LIN {X -45.187,Y 28.575,Z -129.329,A 90.000,B 90.000,C 0.000} C_DIS
LIN {X -45.416,Y 28.575,Z -128.828,A 90.000,B 90.000,C 0.000} C_DIS
LIN {X -45.639,Y 28.575,Z -128.325,A 90.000,B 90.000,C 0.000} C_DIS
LIN {X -46.722,Y 28.575,Z -126.161,A 90.000,B 90.000,C 0.000} C_DIS
LIN {X -47.769,Y 28.575,Z -123.979,A 90.000,B 90.000,C 0.000} C_DIS
LIN {X -48.781,Y 28.575,Z -121.781,A 90.000,B 90.000,C 0.000} C_DIS
LIN {X -144.015,Y 28.575,Z -121.781,A 90.000,B 90.000,C 0.000} C_DIS
LIN {X -144.015,Y 28.575,Z -114.232,A 90.000,B 90.000,C 0.000} C_DIS
LIN {X -53.262,Y 28.575,Z -114.232,A 90.000,B 90.000,C 0.000} C_DIS
LIN {X -53.882,Y 28.575,Z -113.422,A 90.000,B 90.000,C 0.000} C_DIS
LIN {X -54.518,Y 28.575,Z -112.624,A 90.000,B 90.000,C 0.000} C_DIS
LIN {X -56.238,Y 28.575,Z -110.408,A 90.000,B 90.000,C 0.000} C_DIS
LIN {X -57.937,Y 28.575,Z -108.176,A 90.000,B 90.000,C 0.000} C_DIS
LIN {X -59.127,Y 28.575,Z -106.683,A 90.000,B 90.000,C 0.000} C_DIS
LIN {X -144.015,Y 28.575,Z -106.683,A 90.000,B 90.000,C 0.000} C_DIS
LIN {X -144.015,Y 28.575,Z -99.134,A 90.000,B 90.000,C 0.000} C_DIS
LIN {X -64.843,Y 28.575,Z -99.134,A 90.000,B 90.000,C 0.000} C_DIS
LIN {X -65.709,Y 28.575,Z -97.932,A 90.000,B 90.000,C 0.000} C_DIS
LIN {X -66.964,Y 28.575,Z -96.315,A 90.000,B 90.000,C 0.000} C_DIS
LIN {X -68.244,Y 28.575,Z -94.718,A 90.000,B 90.000,C 0.000} C_DIS
LIN {X -69.549,Y 28.575,Z -93.142,A 90.000,B 90.000,C 0.000} C_DIS
LIN {X -70.879,Y 28.575,Z -91.586,A 90.000,B 90.000,C 0.000} C_DIS
LIN {X -144.015,Y 28.575,Z -91.586,A 90.000,B 90.000,C 0.000} C_DIS
LIN {X -144.015,Y 28.575,Z -84.037,A 90.000,B 90.000,C 0.000} C_DIS
LIN {X -77.937,Y 28.575,Z -84.037,A 90.000,B 90.000,C 0.000} C_DIS
LIN {X -78.622,Y 28.575,Z -83.298,A 90.000,B 90.000,C 0.000} C_DIS
LIN {X -79.761,Y 28.575,Z -83.093,A 90.000,B 90.000,C 0.000} C_DIS
LIN {X -80.886,Y 28.575,Z -82.817,A 90.000,B 90.000,C 0.000} C_DIS
LIN {X -81.990,Y 28.575,Z -82.470,A 90.000,B 90.000,C 0.000} C_DIS
LIN {X -83.070,Y 28.575,Z -82.054,A 90.000,B 90.000,C 0.000} C_DIS
LIN {X -84.122,Y 28.575,Z -81.570,A 90.000,B 90.000,C 0.000} C_DIS
LIN {X -85.141,Y 28.575,Z -81.021,A 90.000,B 90.000,C 0.000} C_DIS
LIN {X -86.123,Y 28.575,Z -80.408,A 90.000,B 90.000,C 0.000} C_DIS
LIN {X -87.065,Y 28.575,Z -79.735,A 90.000,B 90.000,C 0.000} C_DIS
LIN {X -87.961,Y 28.575,Z -79.003,A 90.000,B 90.000,C 0.000} C_DIS
LIN {X -88.810,Y 28.575,Z -78.215,A 90.000,B 90.000,C 0.000} C_DIS
LIN {X -89.608,Y 28.575,Z -77.376,A 90.000,B 90.000,C 0.000} C_DIS
LIN {X -90.350,Y 28.575,Z -76.488,A 90.000,B 90.000,C 0.000} C_DIS
LIN {X -144.015,Y 28.575,Z -76.488,A 90.000,B 90.000,C 0.000} C_DIS
LIN {X -144.015,Y 28.575,Z -68.939,A 90.000,B 90.000,C 0.000} C_DIS
LIN {X -94.422,Y 28.575,Z -68.939,A 90.000,B 90.000,C 0.000} C_DIS
LIN {X -95.090,Y 28.575,Z -68.358,A 90.000,B 90.000,C 0.000} C_DIS
LIN {X -95.244,Y 28.575,Z -68.214,A 90.000,B 90.000,C 0.000} C_DIS
LIN {X -95.839,Y 28.575,Z -67.609,A 90.000,B 90.000,C 0.000} C_DIS
LIN {X -96.393,Y 28.575,Z -66.968,A 90.000,B 90.000,C 0.000} C_DIS
LIN {X -96.906,Y 28.575,Z -66.291,A 90.000,B 90.000,C 0.000} C_DIS
LIN {X -97.373,Y 28.575,Z -65.584,A 90.000,B 90.000,C 0.000} C_DIS
LIN {X -97.795,Y 28.575,Z -64.848,A 90.000,B 90.000,C 0.000} C_DIS
LIN {X -98.168,Y 28.575,Z -64.086,A 90.000,B 90.000,C 0.000} C_DIS
LIN {X -99.173,Y 28.575,Z -63.219,A 90.000,B 90.000,C 0.000} C_DIS
LIN {X -100.151,Y 28.575,Z -62.320,A 90.000,B 90.000,C 0.000} C_DIS
LIN {X -101.099,Y 28.575,Z -61.390,A 90.000,B 90.000,C 0.000} C_DIS
LIN {X -144.015,Y 28.575,Z -61.390,A 90.000,B 90.000,C 0.000} C_DIS
LIN {X -144.015,Y 28.575,Z -53.842,A 90.000,B 90.000,C 0.000} C_DIS
LIN {X -106.042,Y 28.575,Z -53.842,A 90.000,B 90.000,C 0.000} C_DIS
LIN {X -106.315,Y 28.575,Z -52.946,A 90.000,B 90.000,C 0.000} C_DIS
LIN {X -106.538,Y 28.575,Z -52.036,A 90.000,B 90.000,C 0.000} C_DIS
LIN {X -106.713,Y 28.575,Z -51.115,A 90.000,B 90.000,C 0.000} C_DIS
LIN {X -106.837,Y 28.575,Z -50.186,A 90.000,B 90.000,C 0.000} C_DIS
LIN {X -106.910,Y 28.575,Z -49.252,A 90.000,B 90.000,C 0.000} C_DIS
LIN {X -106.883,Y 28.575,Z -48.505,A 90.000,B 90.000,C 0.000} C_DIS
LIN {X -106.812,Y 28.575,Z -47.761,A 90.000,B 90.000,C 0.000} C_DIS
LIN {X -106.696,Y 28.575,Z -47.023,A 90.000,B 90.000,C 0.000} C_DIS
LIN {X -106.537,Y 28.575,Z -46.293,A 90.000,B 90.000,C 0.000} C_DIS
LIN {X -144.015,Y 28.575,Z -46.293,A 90.000,B 90.000,C 0.000} C_DIS
LIN {X -144.015,Y 28.575,Z -38.744,A 90.000,B 90.000,C 0.000} C_DIS
LIN {X -101.192,Y 28.575,Z -38.744,A 90.000,B 90.000,C 0.000} C_DIS
LIN {X -144.015,Y 28.575,Z -31.195,A 90.000,B 90.000,C 0.000} C_DIS
LIN {X 98.089,Y 28.575,Z -31.195,A 90.000,B 90.000,C 0.000} C_DIS
LIN {X 99.517,Y 28.575,Z -30.557,A 90.000,B 90.000,C 0.000} C_DIS
LIN {X 100.960,Y 28.575,Z -29.954,A 90.000,B 90.000,C 0.000} C_DIS
LIN {X 102.417,Y 28.575,Z -29.386,A 90.000,B 90.000,C 0.000} C_DIS
LIN {X 103.674,Y 28.575,Z -28.880,A 90.000,B 90.000,C 0.000} C_DIS
LIN {X 104.953,Y 28.575,Z -28.431,A 90.000,B 90.000,C 0.000} C_DIS
LIN {X 106.251,Y 28.575,Z -28.040,A 90.000,B 90.000,C 0.000} C_DIS
LIN {X 107.565,Y 28.575,Z -27.708,A 90.000,B 90.000,C 0.000} C_DIS
LIN {X 108.892,Y 28.575,Z -27.435,A 90.000,B 90.000,C 0.000} C_DIS
LIN {X 109.865,Y 28.575,Z -27.357,A 90.000,B 90.000,C 0.000} C_DIS
LIN {X 110.841,Y 28.575,Z -27.343,A 90.000,B 90.000,C 0.000} C_DIS
LIN {X 111.816,Y 28.575,Z -27.395,A 90.000,B 90.000,C 0.000} C_DIS
LIN {X 112.785,Y 28.575,Z -27.512,A 90.000,B 90.000,C 0.000} C_DIS
LIN {X 113.744,Y 28.575,Z -27.693,A 90.000,B 90.000,C 0.000} C_DIS
LIN {X 114.689,Y 28.575,Z -27.938,A 90.000,B 90.000,C 0.000} C_DIS
LIN {X 114.871,Y 28.575,Z -27.996,A 90.000,B 90.000,C 0.000} C_DIS
LIN {X 115.775,Y 28.575,Z -28.294,A 90.000,B 90.000,C 0.000} C_DIS
LIN {X 116.659,Y 28.575,Z -28.648,A 90.000,B 90.000,C 0.000} C_DIS
LIN {X 117.519,Y 28.575,Z -29.056,A 90.000,B 90.000,C 0.000} C_DIS
LIN {X 118.352,Y 28.575,Z -29.518,A 90.000,B 90.000,C 0.000} C_DIS
LIN {X 118.488,Y 28.575,Z -29.602,A 90.000,B 90.000,C 0.000} C_DIS
LIN {X 119.234,Y 28.575,Z -30.088,A 90.000,B 90.000,C 0.000} C_DIS
LIN {X 119.949,Y 28.575,Z -30.620,A 90.000,B 90.000,C 0.000} C_DIS
LIN {X 120.629,Y 28.575,Z -31.195,A 90.000,B 90.000,C 0.000} C_DIS
LIN {X 144.015,Y 28.575,Z -31.195,A 90.000,B 90.000,C 0.000} C_DIS
LIN {X 144.015,Y 28.575,Z -38.744,A 90.000,B 90.000,C 0.000} C_DIS
LIN {X 125.030,Y 28.575,Z -38.744,A 90.000,B 90.000,C 0.000} C_DIS
LIN {X 125.175,Y 28.575,Z -39.493,A 90.000,B 90.000,C 0.000} C_DIS
LIN {X 125.280,Y 28.575,Z -40.248,A 90.000,B 90.000,C 0.000} C_DIS
LIN {X 125.344,Y 28.575,Z -41.008,A 90.000,B 90.000,C 0.000} C_DIS
LIN {X 125.413,Y 28.575,Z -42.067,A 90.000,B 90.000,C 0.000} C_DIS
LIN {X 125.426,Y 28.575,Z -43.127,A 90.000,B 90.000,C 0.000} C_DIS
LIN {X 125.383,Y 28.575,Z -44.187,A 90.000,B 90.000,C 0.000} C_DIS
LIN {X 125.285,Y 28.575,Z -45.243,A 90.000,B 90.000,C 0.000} C_DIS
LIN {X 125.131,Y 28.575,Z -46.293,A 90.000,B 90.000,C 0.000} C_DIS
LIN {X 144.015,Y 28.575,Z -46.293,A 90.000,B 90.000,C 0.000} C_DIS
LIN {X 144.015,Y 28.575,Z -53.842,A 90.000,B 90.000,C 0.000} C_DIS
LIN {X 122.274,Y 28.575,Z -53.842,A 90.000,B 90.000,C 0.000} C_DIS
LIN {X 121.422,Y 28.575,Z -55.612,A 90.000,B 90.000,C 0.000} C_DIS
LIN {X 120.619,Y 28.575,Z -57.405,A 90.000,B 90.000,C 0.000} C_DIS
LIN {X 119.868,Y 28.575,Z -59.220,A 90.000,B 90.000,C 0.000} C_DIS
LIN {X 119.167,Y 28.575,Z -61.055,A 90.000,B 90.000,C 0.000} C_DIS
LIN {X 119.069,Y 28.575,Z -61.390,A 90.000,B 90.000,C 0.000} C_DIS
LIN {X 144.015,Y 28.575,Z -61.390,A 90.000,B 90.000,C 0.000} C_DIS
LIN {X 144.015,Y 28.575,Z -68.939,A 90.000,B 90.000,C 0.000} C_DIS
LIN {X 116.890,Y 28.575,Z -68.939,A 90.000,B 90.000,C 0.000} C_DIS
LIN {X 116.236,Y 28.575,Z -70.854,A 90.000,B 90.000,C 0.000} C_DIS
LIN {X 115.531,Y 28.575,Z -72.752,A 90.000,B 90.000,C 0.000} C_DIS
LIN {X 114.777,Y 28.575,Z -74.630,A 90.000,B 90.000,C 0.000} C_DIS
LIN {X 113.973,Y 28.575,Z -76.488,A 90.000,B 90.000,C 0.000} C_DIS
LIN {X 144.015,Y 28.575,Z -76.488,A 90.000,B 90.000,C 0.000} C_DIS
LIN {X 144.015,Y 28.575,Z -84.037,A 90.000,B 90.000,C 0.000} C_DIS
LIN {X 110.073,Y 28.575,Z -84.037,A 90.000,B 90.000,C 0.000} C_DIS
LIN {X 109.299,Y 28.575,Z -85.323,A 90.000,B 90.000,C 0.000} C_DIS
LIN {X 108.499,Y 28.575,Z -86.594,A 90.000,B 90.000,C 0.000} C_DIS
LIN {X 107.675,Y 28.575,Z -87.849,A 90.000,B 90.000,C 0.000} C_DIS
LIN {X 107.763,Y 28.575,Z -89.093,A 90.000,B 90.000,C 0.000} C_DIS
LIN {X 107.830,Y 28.575,Z -90.339,A 90.000,B 90.000,C 0.000} C_DIS
LIN {X 107.876,Y 28.575,Z -91.586,A 90.000,B 90.000,C 0.000} C_DIS
LIN {X 144.015,Y 28.575,Z -91.586,A 90.000,B 90.000,C 0.000} C_DIS
LIN {X 144.015,Y 28.575,Z -99.134,A 90.000,B 90.000,C 0.000} C_DIS
LIN {X 107.706,Y 28.575,Z -99.134,A 90.000,B 90.000,C 0.000} C_DIS
LIN {X 107.629,Y 28.575,Z -100.093,A 90.000,B 90.000,C 0.000} C_DIS
LIN {X 107.540,Y 28.575,Z -101.051,A 90.000,B 90.000,C 0.000} C_DIS
LIN {X 107.480,Y 28.575,Z -102.572,A 90.000,B 90.000,C 0.000} C_DIS
LIN {X 107.467,Y 28.575,Z -102.703,A 90.000,B 90.000,C 0.000} C_DIS
LIN {X 107.463,Y 28.575,Z -103.506,A 90.000,B 90.000,C 0.000} C_DIS
LIN {X 107.504,Y 28.575,Z -104.308,A 90.000,B 90.000,C 0.000} C_DIS
LIN {X 107.589,Y 28.575,Z -105.106,A 90.000,B 90.000,C 0.000} C_DIS
LIN {X 107.718,Y 28.575,Z -105.899,A 90.000,B 90.000,C 0.000} C_DIS
LIN {X 107.891,Y 28.575,Z -106.683,A 90.000,B 90.000,C 0.000} C_DIS
LIN {X 144.015,Y 28.575,Z -106.683,A 90.000,B 90.000,C 0.000} C_DIS
LIN {X 144.015,Y 28.575,Z -114.232,A 90.000,B 90.000,C 0.000} C_DIS
LIN {X 108.666,Y 28.575,Z -114.232,A 90.000,B 90.000,C 0.000} C_DIS
LIN {X 108.827,Y 28.575,Z -116.746,A 90.000,B 90.000,C 0.000} C_DIS
LIN {X 108.950,Y 28.575,Z -119.263,A 90.000,B 90.000,C 0.000} C_DIS
LIN {X 109.037,Y 28.575,Z -121.781,A 90.000,B 90.000,C 0.000} C_DIS
LIN {X 144.015,Y 28.575,Z -121.781,A 90.000,B 90.000,C 0.000} C_DIS
LIN {X 144.015,Y 28.575,Z -129.329,A 90.000,B 90.000,C 0.000} C_DIS
LIN {X 109.075,Y 28.575,Z -129.329,A 90.000,B 90.000,C 0.000} C_DIS
LIN {X 109.014,Y 28.575,Z -131.847,A 90.000,B 90.000,C 0.000} C_DIS
LIN {X 108.916,Y 28.575,Z -134.363,A 90.000,B 90.000,C 0.000} C_DIS
LIN {X 108.782,Y 28.575,Z -136.878,A 90.000,B 90.000,C 0.000} C_DIS
LIN {X 144.015,Y 28.575,Z -136.878,A 90.000,B 90.000,C 0.000} C_DIS
LIN {X 144.015,Y 28.575,Z -144.427,A 90.000,B 90.000,C 0.000} C_DIS
LIN {X 108.182,Y 28.575,Z -144.427,A 90.000,B 90.000,C 0.000} C_DIS
LIN {X 107.856,Y 28.575,Z -148.203,A 90.000,B 90.000,C 0.000} C_DIS
LIN {X 107.490,Y 28.575,Z -151.976,A 90.000,B 90.000,C 0.000} C_DIS
LIN {X 144.015,Y 28.575,Z -151.976,A 90.000,B 90.000,C 0.000} C_DIS
LIN {X 144.015,Y 28.575,Z -159.525,A 90.000,B 90.000,C 0.000} C_DIS
LIN {X 106.632,Y 28.575,Z -159.525,A 90.000,B 90.000,C 0.000} C_DIS
LIN {X 106.141,Y 28.575,Z -163.302,A 90.000,B 90.000,C 0.000} C_DIS
LIN {X 105.608,Y 28.575,Z -167.073,A 90.000,B 90.000,C 0.000} C_DIS
LIN {X 144.015,Y 28.575,Z -167.073,A 90.000,B 90.000,C 0.000} C_DIS
LIN {X 144.015,Y 28.575,Z -174.622,A 90.000,B 90.000,C 0.000} C_DIS
LIN {X 104.436,Y 28.575,Z -174.622,A 90.000,B 90.000,C 0.000} C_DIS
LIN {X 104.078,Y 28.575,Z -177.133,A 90.000,B 90.000,C 0.000} C_DIS
LIN {X 103.757,Y 28.575,Z -179.650,A 90.000,B 90.000,C 0.000} C_DIS
LIN {X 103.474,Y 28.575,Z -182.171,A 90.000,B 90.000,C 0.000} C_DIS
LIN {X 144.015,Y 28.575,Z -182.171,A 90.000,B 90.000,C 0.000} C_DIS
LIN {X 144.015,Y 28.575,Z -189.720,A 90.000,B 90.000,C 0.000} C_DIS
LIN {X 102.854,Y 28.575,Z -189.720,A 90.000,B 90.000,C 0.000} C_DIS
LIN {X 102.786,Y 28.575,Z -190.930,A 90.000,B 90.000,C 0.000} C_DIS
LIN {X 102.727,Y 28.575,Z -192.140,A 90.000,B 90.000,C 0.000} C_DIS
LIN {X 102.588,Y 28.575,Z -193.853,A 90.000,B 90.000,C 0.000} C_DIS
LIN {X 102.412,Y 28.575,Z -195.563,A 90.000,B 90.000,C 0.000} C_DIS
LIN {X 102.197,Y 28.575,Z -197.269,A 90.000,B 90.000,C 0.000} C_DIS
LIN {X 144.015,Y 28.575,Z -197.269,A 90.000,B 90.000,C 0.000} C_DIS
LIN {X 144.015,Y 28.575,Z -204.817,A 90.000,B 90.000,C 0.000} C_DIS
LIN {X 100.774,Y 28.575,Z -204.817,A 90.000,B 90.000,C 0.000} C_DIS
LIN {X 100.506,Y 28.575,Z -205.895,A 90.000,B 90.000,C 0.000} C_DIS
LIN {X 100.223,Y 28.575,Z -206.969,A 90.000,B 90.000,C 0.000} C_DIS
LIN {X 99.604,Y 28.575,Z -209.358,A 90.000,B 90.000,C 0.000} C_DIS
LIN {X 99.003,Y 28.575,Z -211.751,A 90.000,B 90.000,C 0.000} C_DIS
LIN {X 98.837,Y 28.575,Z -212.366,A 90.000,B 90.000,C 0.000} C_DIS
LIN {X 144.015,Y 28.575,Z -212.366,A 90.000,B 90.000,C 0.000} C_DIS
LIN {X 144.015,Y 28.575,Z -219.915,A 90.000,B 90.000,C 0.000} C_DIS
LIN {X 96.861,Y 28.575,Z -219.915,A 90.000,B 90.000,C 0.000} C_DIS
LIN {X 95.882,Y 28.575,Z -223.687,A 90.000,B 90.000,C 0.000} C_DIS
LIN {X 94.920,Y 28.575,Z -227.464,A 90.000,B 90.000,C 0.000} C_DIS
LIN {X 144.015,Y 28.575,Z -227.464,A 90.000,B 90.000,C 0.000} C_DIS
LIN {X 144.015,Y 28.575,Z -235.012,A 90.000,B 90.000,C 0.000} C_DIS
LIN {X 92.952,Y 28.575,Z -235.012,A 90.000,B 90.000,C 0.000} C_DIS
LIN {X 92.216,Y 28.575,Z -237.541,A 90.000,B 90.000,C 0.000} C_DIS
LIN {X 91.439,Y 28.575,Z -240.057,A 90.000,B 90.000,C 0.000} C_DIS
LIN {X 90.622,Y 28.575,Z -242.561,A 90.000,B 90.000,C 0.000} C_DIS
LIN {X 144.015,Y 28.575,Z -242.561,A 90.000,B 90.000,C 0.000} C_DIS
LIN {X 144.015,Y 28.575,Z -23.646,A 90.000,B 90.000,C 0.000} C_DIS
LIN {X -144.015,Y 28.575,Z -23.646,A 90.000,B 90.000,C 0.000} C_DIS
LIN {X -144.015,Y 28.575,Z -16.098,A 90.000,B 90.000,C 0.000} C_DIS
LIN {X 144.015,Y 28.575,Z -16.098,A 90.000,B 90.000,C 0.000} C_DIS
LIN {X 144.015,Y 28.575,Z -8.549,A 90.000,B 90.000,C 0.000} C_DIS
LIN {X -144.015,Y 28.575,Z -8.549,A 90.000,B 90.000,C 0.000} C_DIS
LIN {X -144.015,Y 28.575,Z -1.000,A 90.000,B 90.000,C 0.000} C_DIS
LIN {X 144.015,Y 28.575,Z -1.000,A 90.000,B 90.000,C 0.000} C_DIS
LIN {X 29.140,Y 28.575,Z -36.338,A 90.000,B 90.000,C 0.000} C_DIS
LIN {X 27.794,Y 28.575,Z -36.582,A 90.000,B 90.000,C 0.000} C_DIS
LIN {X 26.460,Y 28.575,Z -36.890,A 90.000,B 90.000,C 0.000} C_DIS
LIN {X 25.143,Y 28.575,Z -37.261,A 90.000,B 90.000,C 0.000} C_DIS
LIN {X 23.845,Y 28.575,Z -37.694,A 90.000,B 90.000,C 0.000} C_DIS
LIN {X 22.570,Y 28.575,Z -38.189,A 90.000,B 90.000,C 0.000} C_DIS
LIN {X 21.319,Y 28.575,Z -38.744,A 90.000,B 90.000,C 0.000} C_DIS
LIN {X -57.409,Y 28.575,Z -38.744,A 90.000,B 90.000,C 0.000} C_DIS
LIN {X 21.319,Y 28.575,Z -38.744,A 90.000,B 90.000,C 0.000} C_DIS
LIN {X 22.459,Y 28.575,Z -38.235,A 90.000,B 90.000,C 0.000} C_DIS
LIN {X 23.620,Y 28.575,Z -37.777,A 90.000,B 90.000,C 0.000} C_DIS
LIN {X 24.800,Y 28.575,Z -37.369,A 90.000,B 90.000,C 0.000} C_DIS
LIN {X 25.996,Y 28.575,Z -37.013,A 90.000,B 90.000,C 0.000} C_DIS
LIN {X 27.207,Y 28.575,Z -36.709,A 90.000,B 90.000,C 0.000} C_DIS
LIN {X 28.430,Y 28.575,Z -36.459,A 90.000,B 90.000,C 0.000} C_DIS
LIN {X 29.663,Y 28.575,Z -36.261,A 90.000,B 90.000,C 0.000} C_DIS
LIN {X 30.903,Y 28.575,Z -36.117,A 90.000,B 90.000,C 0.000} C_DIS
LIN {X 31.600,Y 28.575,Z -35.921,A 90.000,B 90.000,C 0.000} C_DIS
LIN {X 32.288,Y 28.575,Z -35.694,A 90.000,B 90.000,C 0.000} C_DIS
LIN {X 32.964,Y 28.575,Z -35.437,A 90.000,B 90.000,C 0.000} C_DIS
LIN {X 33.629,Y 28.575,Z -35.149,A 90.000,B 90.000,C 0.000} C_DIS
LIN {X 34.932,Y 28.575,Z -34.685,A 90.000,B 90.000,C 0.000} C_DIS
LIN {X 36.256,Y 28.575,Z -34.283,A 90.000,B 90.000,C 0.000} C_DIS
LIN {X 37.598,Y 28.575,Z -33.944,A 90.000,B 90.000,C 0.000} C_DIS
LIN {X 38.954,Y 28.575,Z -33.669,A 90.000,B 90.000,C 0.000} C_DIS
LIN {X 40.321,Y 28.575,Z -33.458,A 90.000,B 90.000,C 0.000} C_DIS
LIN {X 41.697,Y 28.575,Z -33.311,A 90.000,B 90.000,C 0.000} C_DIS
LIN {X 43.078,Y 28.575,Z -33.230,A 90.000,B 90.000,C 0.000} C_DIS
LIN {X 44.461,Y 28.575,Z -33.214,A 90.000,B 90.000,C 0.000} C_DIS
LIN {X 45.844,Y 28.575,Z -33.263,A 90.000,B 90.000,C 0.000} C_DIS
LIN {X 47.223,Y 28.575,Z -33.377,A 90.000,B 90.000,C 0.000} C_DIS
LIN {X 48.277,Y 28.575,Z -33.536,A 90.000,B 90.000,C 0.000} C_DIS
LIN {X 49.321,Y 28.575,Z -33.745,A 90.000,B 90.000,C 0.000} C_DIS
LIN {X 50.355,Y 28.575,Z -34.002,A 90.000,B 90.000,C 0.000} C_DIS
LIN {X 51.376,Y 28.575,Z -34.308,A 90.000,B 90.000,C 0.000} C_DIS
LIN {X 52.381,Y 28.575,Z -34.661,A 90.000,B 90.000,C 0.000} C_DIS
LIN {X 53.368,Y 28.575,Z -35.062,A 90.000,B 90.000,C 0.000} C_DIS
LIN {X 54.336,Y 28.575,Z -35.508,A 90.000,B 90.000,C 0.000} C_DIS
LIN {X 55.757,Y 28.575,Z -36.249,A 90.000,B 90.000,C 0.000} C_DIS
LIN {X 57.152,Y 28.575,Z -37.036,A 90.000,B 90.000,C 0.000} C_DIS
LIN {X 58.521,Y 28.575,Z -37.868,A 90.000,B 90.000,C 0.000} C_DIS
LIN {X 59.863,Y 28.575,Z -38.744,A 90.000,B 90.000,C 0.000} C_DIS
LIN {X 85.593,Y 28.575,Z -38.744,A 90.000,B 90.000,C 0.000} C_DIS
LIN {X 84.432,Y 28.575,Z -39.691,A 90.000,B 90.000,C 0.000} C_DIS
LIN {X 83.310,Y 28.575,Z -40.684,A 90.000,B 90.000,C 0.000} C_DIS
LIN {X 82.231,Y 28.575,Z -41.723,A 90.000,B 90.000,C 0.000} C_DIS
LIN {X 81.194,Y 28.575,Z -42.805,A 90.000,B 90.000,C 0.000} C_DIS
LIN {X 80.203,Y 28.575,Z -43.929,A 90.000,B 90.000,C 0.000} C_DIS
LIN {X 79.259,Y 28.575,Z -45.092,A 90.000,B 90.000,C 0.000} C_DIS
LIN {X 78.363,Y 28.575,Z -46.293,A 90.000,B 90.000,C 0.000} C_DIS
LIN {X 68.870,Y 28.575,Z -46.293,A 90.000,B 90.000,C 0.000} C_DIS
LIN {X 69.482,Y 28.575,Z -48.217,A 90.000,B 90.000,C 0.000} C_DIS
LIN {X 66.563,Y 28.575,Z -45.535,A 90.000,B 90.000,C 0.000} C_DIS
LIN {X 63.627,Y 28.575,Z -42.871,A 90.000,B 90.000,C 0.000} C_DIS
LIN {X 62.337,Y 28.575,Z -41.805,A 90.000,B 90.000,C 0.000} C_DIS
LIN {X 61.011,Y 28.575,Z -40.784,A 90.000,B 90.000,C 0.000} C_DIS
LIN {X 59.650,Y 28.575,Z -39.810,A 90.000,B 90.000,C 0.000} C_DIS
LIN {X 58.256,Y 28.575,Z -38.884,A 90.000,B 90.000,C 0.000} C_DIS
LIN {X 56.830,Y 28.575,Z -38.007,A 90.000,B 90.000,C 0.000} C_DIS
LIN {X 55.375,Y 28.575,Z -37.180,A 90.000,B 90.000,C 0.000} C_DIS
LIN {X 53.892,Y 28.575,Z -36.404,A 90.000,B 90.000,C 0.000} C_DIS
LIN {X 52.813,Y 28.575,Z -35.912,A 90.000,B 90.000,C 0.000} C_DIS
LIN {X 51.709,Y 28.575,Z -35.479,A 90.000,B 90.000,C 0.000} C_DIS
LIN {X 50.583,Y 28.575,Z -35.108,A 90.000,B 90.000,C 0.000} C_DIS
LIN {X 49.439,Y 28.575,Z -34.799,A 90.000,B 90.000,C 0.000} C_DIS
LIN {X 48.279,Y 28.575,Z -34.553,A 90.000,B 90.000,C 0.000} C_DIS
LIN {X 47.107,Y 28.575,Z -34.370,A 90.000,B 90.000,C 0.000} C_DIS
LIN {X 45.779,Y 28.575,Z -34.260,A 90.000,B 90.000,C 0.000} C_DIS
LIN {X 44.448,Y 28.575,Z -34.213,A 90.000,B 90.000,C 0.000} C_DIS
LIN {X 43.116,Y 28.575,Z -34.229,A 90.000,B 90.000,C 0.000} C_DIS
LIN {X 41.786,Y 28.575,Z -34.307,A 90.000,B 90.000,C 0.000} C_DIS
LIN {X 40.461,Y 28.575,Z -34.448,A 90.000,B 90.000,C 0.000} C_DIS
LIN {X 39.144,Y 28.575,Z -34.651,A 90.000,B 90.000,C 0.000} C_DIS
LIN {X 37.839,Y 28.575,Z -34.915,A 90.000,B 90.000,C 0.000} C_DIS
LIN {X 36.547,Y 28.575,Z -35.241,A 90.000,B 90.000,C 0.000} C_DIS
LIN {X 35.271,Y 28.575,Z -35.626,A 90.000,B 90.000,C 0.000} C_DIS
LIN {X 34.016,Y 28.575,Z -36.072,A 90.000,B 90.000,C 0.000} C_DIS
LIN {X 33.299,Y 28.575,Z -36.381,A 90.000,B 90.000,C 0.000} C_DIS
LIN {X 32.568,Y 28.575,Z -36.657,A 90.000,B 90.000,C 0.000} C_DIS
LIN {X 31.826,Y 28.575,Z -36.899,A 90.000,B 90.000,C 0.000} C_DIS
LIN {X 31.073,Y 28.575,Z -37.106,A 90.000,B 90.000,C 0.000} C_DIS
LIN {X 29.699,Y 28.575,Z -37.266,A 90.000,B 90.000,C 0.000} C_DIS
LIN {X 28.336,Y 28.575,Z -37.493,A 90.000,B 90.000,C 0.000} C_DIS
LIN {X 26.985,Y 28.575,Z -37.789,A 90.000,B 90.000,C 0.000} C_DIS
LIN {X 25.650,Y 28.575,Z -38.152,A 90.000,B 90.000,C 0.000} C_DIS
LIN {X 24.336,Y 28.575,Z -38.581,A 90.000,B 90.000,C 0.000} C_DIS
LIN {X 23.044,Y 28.575,Z -39.075,A 90.000,B 90.000,C 0.000} C_DIS
LIN {X 21.779,Y 28.575,Z -39.632,A 90.000,B 90.000,C 0.000} C_DIS
LIN {X 20.543,Y 28.575,Z -40.253,A 90.000,B 90.000,C 0.000} C_DIS
LIN {X 19.340,Y 28.575,Z -40.934,A 90.000,B 90.000,C 0.000} C_DIS
LIN {X 19.220,Y 28.575,Z -40.990,A 90.000,B 90.000,C 0.000} C_DIS
LIN {X 18.259,Y 28.575,Z -41.521,A 90.000,B 90.000,C 0.000} C_DIS
LIN {X 17.326,Y 28.575,Z -42.099,A 90.000,B 90.000,C 0.000} C_DIS
LIN {X 16.423,Y 28.575,Z -42.722,A 90.000,B 90.000,C 0.000} C_DIS
LIN {X 15.552,Y 28.575,Z -43.390,A 90.000,B 90.000,C 0.000} C_DIS
LIN {X 14.715,Y 28.575,Z -44.100,A 90.000,B 90.000,C 0.000} C_DIS
LIN {X 13.914,Y 28.575,Z -44.850,A 90.000,B 90.000,C 0.000} C_DIS
LIN {X 13.152,Y 28.575,Z -45.640,A 90.000,B 90.000,C 0.000} C_DIS
LIN {X 12.442,Y 28.575,Z -45.473,A 90.000,B 90.000,C 0.000} C_DIS
LIN {X 11.722,Y 28.575,Z -45.350,A 90.000,B 90.000,C 0.000} C_DIS
LIN {X 10.997,Y 28.575,Z -45.271,A 90.000,B 90.000,C 0.000} C_DIS
LIN {X 8.986,Y 28.575,Z -45.256,A 90.000,B 90.000,C 0.000} C_DIS
LIN {X 6.975,Y 28.575,Z -45.267,A 90.000,B 90.000,C 0.000} C_DIS
LIN {X 4.964,Y 28.575,Z -45.305,A 90.000,B 90.000,C 0.000} C_DIS
LIN {X 1.301,Y 28.575,Z -44.995,A 90.000,B 90.000,C 0.000} C_DIS
LIN {X -2.365,Y 28.575,Z -44.725,A 90.000,B 90.000,C 0.000} C_DIS
LIN {X -3.978,Y 28.575,Z -44.551,A 90.000,B 90.000,C 0.000} C_DIS
LIN {X -5.596,Y 28.575,Z -44.438,A 90.000,B 90.000,C 0.000} C_DIS
LIN {X -7.218,Y 28.575,Z -44.386,A 90.000,B 90.000,C 0.000} C_DIS
LIN {X -8.840,Y 28.575,Z -44.395,A 90.000,B 90.000,C 0.000} C_DIS
LIN {X -10.460,Y 28.575,Z -44.464,A 90.000,B 90.000,C 0.000} C_DIS
LIN {X -12.077,Y 28.575,Z -44.595,A 90.000,B 90.000,C 0.000} C_DIS
LIN {X -13.688,Y 28.575,Z -44.786,A 90.000,B 90.000,C 0.000} C_DIS
LIN {X -15.291,Y 28.575,Z -45.038,A 90.000,B 90.000,C 0.000} C_DIS
LIN {X -16.883,Y 28.575,Z -45.349,A 90.000,B 90.000,C 0.000} C_DIS
LIN {X -19.176,Y 28.575,Z -46.115,A 90.000,B 90.000,C 0.000} C_DIS
LIN {X -21.472,Y 28.575,Z -46.874,A 90.000,B 90.000,C 0.000} C_DIS
LIN {X -21.555,Y 28.575,Z -46.895,A 90.000,B 90.000,C 0.000} C_DIS
LIN {X -22.240,Y 28.575,Z -46.779,A 90.000,B 90.000,C 0.000} C_DIS
LIN {X -22.922,Y 28.575,Z -46.640,A 90.000,B 90.000,C 0.000} C_DIS
LIN {X -23.598,Y 28.575,Z -46.480,A 90.000,B 90.000,C 0.000} C_DIS
LIN {X -26.728,Y 28.575,Z -45.653,A 90.000,B 90.000,C 0.000} C_DIS
LIN {X -29.872,Y 28.575,Z -44.883,A 90.000,B 90.000,C 0.000} C_DIS
LIN {X -33.030,Y 28.575,Z -44.169,A 90.000,B 90.000,C 0.000} C_DIS
LIN {X -36.199,Y 28.575,Z -43.512,A 90.000,B 90.000,C 0.000} C_DIS
LIN {X -39.380,Y 28.575,Z -42.912,A 90.000,B 90.000,C 0.000} C_DIS
LIN {X -42.572,Y 28.575,Z -42.370,A 90.000,B 90.000,C 0.000} C_DIS
LIN {X -46.004,Y 28.575,Z -41.968,A 90.000,B 90.000,C 0.000} C_DIS
LIN {X -49.434,Y 28.575,Z -41.541,A 90.000,B 90.000,C 0.000} C_DIS
LIN {X -52.860,Y 28.575,Z -41.088,A 90.000,B 90.000,C 0.000} C_DIS
LIN {X -54.547,Y 28.575,Z -40.655,A 90.000,B 90.000,C 0.000} C_DIS
LIN {X -56.220,Y 28.575,Z -40.172,A 90.000,B 90.000,C 0.000} C_DIS
LIN {X -57.879,Y 28.575,Z -39.642,A 90.000,B 90.000,C 0.000} C_DIS
LIN {X -59.521,Y 28.575,Z -39.063,A 90.000,B 90.000,C 0.000} C_DIS
LIN {X -61.146,Y 28.575,Z -38.436,A 90.000,B 90.000,C 0.000} C_DIS
LIN {X -62.814,Y 28.575,Z -37.607,A 90.000,B 90.000,C 0.000} C_DIS
LIN {X -64.507,Y 28.575,Z -36.832,A 90.000,B 90.000,C 0.000} C_DIS
LIN {X -66.224,Y 28.575,Z -36.111,A 90.000,B 90.000,C 0.000} C_DIS
LIN {X -67.963,Y 28.575,Z -35.445,A 90.000,B 90.000,C 0.000} C_DIS
LIN {X -69.722,Y 28.575,Z -34.835,A 90.000,B 90.000,C 0.000} C_DIS
LIN {X -71.499,Y 28.575,Z -34.280,A 90.000,B 90.000,C 0.000} C_DIS
LIN {X -73.294,Y 28.575,Z -33.783,A 90.000,B 90.000,C 0.000} C_DIS
LIN {X -74.373,Y 28.575,Z -33.417,A 90.000,B 90.000,C 0.000} C_DIS
LIN {X -75.472,Y 28.575,Z -33.118,A 90.000,B 90.000,C 0.000} C_DIS
LIN {X -76.588,Y 28.575,Z -32.887,A 90.000,B 90.000,C 0.000} C_DIS
LIN {X -77.715,Y 28.575,Z -32.725,A 90.000,B 90.000,C 0.000} C_DIS
LIN {X -78.851,Y 28.575,Z -32.632,A 90.000,B 90.000,C 0.000} C_DIS
LIN {X -79.989,Y 28.575,Z -32.609,A 90.000,B 90.000,C 0.000} C_DIS
LIN {X -81.128,Y 28.575,Z -32.655,A 90.000,B 90.000,C 0.000} C_DIS
LIN {X -82.261,Y 28.575,Z -32.771,A 90.000,B 90.000,C 0.000} C_DIS
LIN {X -83.165,Y 28.575,Z -33.000,A 90.000,B 90.000,C 0.000} C_DIS
LIN {X -84.049,Y 28.575,Z -33.295,A 90.000,B 90.000,C 0.000} C_DIS
LIN {X -84.909,Y 28.575,Z -33.655,A 90.000,B 90.000,C 0.000} C_DIS
LIN {X -85.740,Y 28.575,Z -34.077,A 90.000,B 90.000,C 0.000} C_DIS
LIN {X -86.538,Y 28.575,Z -34.560,A 90.000,B 90.000,C 0.000} C_DIS
LIN {X -87.297,Y 28.575,Z -35.100,A 90.000,B 90.000,C 0.000} C_DIS
LIN {X -88.015,Y 28.575,Z -35.695,A 90.000,B 90.000,C 0.000} C_DIS
LIN {X -88.687,Y 28.575,Z -36.341,A 90.000,B 90.000,C 0.000} C_DIS
LIN {X -89.309,Y 28.575,Z -37.036,A 90.000,B 90.000,C 0.000} C_DIS
LIN {X -89.878,Y 28.575,Z -37.774,A 90.000,B 90.000,C 0.000} C_DIS
LIN {X -90.649,Y 28.575,Z -37.631,A 90.000,B 90.000,C 0.000} C_DIS
LIN {X -91.426,Y 28.575,Z -37.528,A 90.000,B 90.000,C 0.000} C_DIS
LIN {X -92.207,Y 28.575,Z -37.464,A 90.000,B 90.000,C 0.000} C_DIS
LIN {X -92.991,Y 28.575,Z -37.439,A 90.000,B 90.000,C 0.000} C_DIS
LIN {X -93.775,Y 28.575,Z -37.454,A 90.000,B 90.000,C 0.000} C_DIS
LIN {X -94.640,Y 28.575,Z -37.482,A 90.000,B 90.000,C 0.000} C_DIS
LIN {X -95.500,Y 28.575,Z -37.572,A 90.000,B 90.000,C 0.000} C_DIS
LIN {X -96.352,Y 28.575,Z -37.724,A 90.000,B 90.000,C 0.000} C_DIS
LIN {X -97.191,Y 28.575,Z -37.937,A 90.000,B 90.000,C 0.000} C_DIS
LIN {X -98.012,Y 28.575,Z -38.210,A 90.000,B 90.000,C 0.000} C_DIS
LIN {X -98.812,Y 28.575,Z -38.541,A 90.000,B 90.000,C 0.000} C_DIS
LIN {X -99.585,Y 28.575,Z -38.928,A 90.000,B 90.000,C 0.000} C_DIS
LIN {X -100.329,Y 28.575,Z -39.370,A 90.000,B 90.000,C 0.000} C_DIS
LIN {X -101.039,Y 28.575,Z -39.865,A 90.000,B 90.000,C 0.000} C_DIS
LIN {X -101.712,Y 28.575,Z -40.409,A 90.000,B 90.000,C 0.000} C_DIS
LIN {X -101.798,Y 28.575,Z -40.488,A 90.000,B 90.000,C 0.000} C_DIS
LIN {X -102.248,Y 28.575,Z -40.851,A 90.000,B 90.000,C 0.000} C_DIS
LIN {X -102.663,Y 28.575,Z -41.255,A 90.000,B 90.000,C 0.000} C_DIS
LIN {X -103.037,Y 28.575,Z -41.696,A 90.000,B 90.000,C 0.000} C_DIS
LIN {X -103.112,Y 28.575,Z -41.797,A 90.000,B 90.000,C 0.000} C_DIS
LIN {X -103.673,Y 28.575,Z -42.501,A 90.000,B 90.000,C 0.000} C_DIS
LIN {X -104.177,Y 28.575,Z -43.248,A 90.000,B 90.000,C 0.000} C_DIS
LIN {X -104.622,Y 28.575,Z -44.031,A 90.000,B 90.000,C 0.000} C_DIS
LIN {X -105.004,Y 28.575,Z -44.846,A 90.000,B 90.000,C 0.000} C_DIS
LIN {X -105.321,Y 28.575,Z -45.689,A 90.000,B 90.000,C 0.000} C_DIS
LIN {X -105.572,Y 28.575,Z -46.554,A 90.000,B 90.000,C 0.000} C_DIS
LIN {X -105.754,Y 28.575,Z -47.436,A 90.000,B 90.000,C 0.000} C_DIS
LIN {X -105.867,Y 28.575,Z -48.329,A 90.000,B 90.000,C 0.000} C_DIS
LIN {X -105.910,Y 28.575,Z -49.229,A 90.000,B 90.000,C 0.000} C_DIS
LIN {X -105.825,Y 28.575,Z -50.238,A 90.000,B 90.000,C 0.000} C_DIS
LIN {X -105.677,Y 28.575,Z -51.241,A 90.000,B 90.000,C 0.000} C_DIS
LIN {X -105.467,Y 28.575,Z -52.232,A 90.000,B 90.000,C 0.000} C_DIS
LIN {X -105.196,Y 28.575,Z -53.208,A 90.000,B 90.000,C 0.000} C_DIS
LIN {X -104.865,Y 28.575,Z -54.165,A 90.000,B 90.000,C 0.000} C_DIS
LIN {X -104.475,Y 28.575,Z -55.100,A 90.000,B 90.000,C 0.000} C_DIS
LIN {X -104.027,Y 28.575,Z -56.009,A 90.000,B 90.000,C 0.000} C_DIS
LIN {X -103.525,Y 28.575,Z -56.888,A 90.000,B 90.000,C 0.000} C_DIS
LIN {X -102.968,Y 28.575,Z -57.735,A 90.000,B 90.000,C 0.000} C_DIS
LIN {X -102.360,Y 28.575,Z -58.545,A 90.000,B 90.000,C 0.000} C_DIS
LIN {X -102.236,Y 28.575,Z -58.691,A 90.000,B 90.000,C 0.000} C_DIS
LIN {X -101.323,Y 28.575,Z -59.710,A 90.000,B 90.000,C 0.000} C_DIS
LIN {X -100.376,Y 28.575,Z -60.699,A 90.000,B 90.000,C 0.000} C_DIS
LIN {X -99.398,Y 28.575,Z -61.655,A 90.000,B 90.000,C 0.000} C_DIS
LIN {X -98.387,Y 28.575,Z -62.578,A 90.000,B 90.000,C 0.000} C_DIS
LIN {X -97.347,Y 28.575,Z -63.467,A 90.000,B 90.000,C 0.000} C_DIS
LIN {X -96.999,Y 28.575,Z -64.210,A 90.000,B 90.000,C 0.000} C_DIS
LIN {X -96.601,Y 28.575,Z -64.928,A 90.000,B 90.000,C 0.000} C_DIS
LIN {X -96.156,Y 28.575,Z -65.618,A 90.000,B 90.000,C 0.000} C_DIS
LIN {X -95.666,Y 28.575,Z -66.276,A 90.000,B 90.000,C 0.000} C_DIS
LIN {X -95.132,Y 28.575,Z -66.900,A 90.000,B 90.000,C 0.000} C_DIS
LIN {X -94.558,Y 28.575,Z -67.487,A 90.000,B 90.000,C 0.000} C_DIS
LIN {X -94.418,Y 28.575,Z -67.617,A 90.000,B 90.000,C 0.000} C_DIS
LIN {X -93.476,Y 28.575,Z -68.431,A 90.000,B 90.000,C 0.000} C_DIS
LIN {X -92.517,Y 28.575,Z -69.225,A 90.000,B 90.000,C 0.000} C_DIS
LIN {X -92.335,Y 28.575,Z -70.071,A 90.000,B 90.000,C 0.000} C_DIS
LIN {X -92.109,Y 28.575,Z -70.907,A 90.000,B 90.000,C 0.000} C_DIS
LIN {X -91.840,Y 28.575,Z -71.729,A 90.000,B 90.000,C 0.000} C_DIS
LIN {X -91.529,Y 28.575,Z -72.537,A 90.000,B 90.000,C 0.000} C_DIS
LIN {X -91.177,Y 28.575,Z -73.328,A 90.000,B 90.000,C 0.000} C_DIS
LIN {X -90.784,Y 28.575,Z -74.099,A 90.000,B 90.000,C 0.000} C_DIS
LIN {X -90.680,Y 28.575,Z -74.266,A 90.000,B 90.000,C 0.000} C_DIS
LIN {X -90.073,Y 28.575,Z -75.186,A 90.000,B 90.000,C 0.000} C_DIS
LIN {X -89.408,Y 28.575,Z -76.066,A 90.000,B 90.000,C 0.000} C_DIS
LIN {X -88.688,Y 28.575,Z -76.901,A 90.000,B 90.000,C 0.000} C_DIS
LIN {X -87.917,Y 28.575,Z -77.689,A 90.000,B 90.000,C 0.000} C_DIS
LIN {X -87.097,Y 28.575,Z -78.426,A 90.000,B 90.000,C 0.000} C_DIS
LIN {X -86.232,Y 28.575,Z -79.109,A 90.000,B 90.000,C 0.000} C_DIS
LIN {X -85.325,Y 28.575,Z -79.736,A 90.000,B 90.000,C 0.000} C_DIS
LIN {X -84.380,Y 28.575,Z -80.303,A 90.000,B 90.000,C 0.000} C_DIS
LIN {X -83.400,Y 28.575,Z -80.810,A 90.000,B 90.000,C 0.000} C_DIS
LIN {X -82.390,Y 28.575,Z -81.252,A 90.000,B 90.000,C 0.000} C_DIS
LIN {X -81.354,Y 28.575,Z -81.629,A 90.000,B 90.000,C 0.000} C_DIS
LIN {X -80.296,Y 28.575,Z -81.940,A 90.000,B 90.000,C 0.000} C_DIS
LIN {X -79.221,Y 28.575,Z -82.182,A 90.000,B 90.000,C 0.000} C_DIS
LIN {X -78.132,Y 28.575,Z -82.356,A 90.000,B 90.000,C 0.000} C_DIS
LIN {X -76.717,Y 28.575,Z -83.880,A 90.000,B 90.000,C 0.000} C_DIS
LIN {X -74.918,Y 28.575,Z -85.702,A 90.000,B 90.000,C 0.000} C_DIS
LIN {X -73.156,Y 28.575,Z -87.558,A 90.000,B 90.000,C 0.000} C_DIS
LIN {X -71.429,Y 28.575,Z -89.449,A 90.000,B 90.000,C 0.000} C_DIS
LIN {X -69.741,Y 28.575,Z -91.373,A 90.000,B 90.000,C 0.000} C_DIS
LIN {X -68.090,Y 28.575,Z -93.329,A 90.000,B 90.000,C 0.000} C_DIS
LIN {X -66.477,Y 28.575,Z -95.317,A 90.000,B 90.000,C 0.000} C_DIS
LIN {X -64.904,Y 28.575,Z -97.337,A 90.000,B 90.000,C 0.000} C_DIS
LIN {X -63.019,Y 28.575,Z -99.934,A 90.000,B 90.000,C 0.000} C_DIS
LIN {X -61.098,Y 28.575,Z -102.504,A 90.000,B 90.000,C 0.000} C_DIS
LIN {X -59.140,Y 28.575,Z -105.046,A 90.000,B 90.000,C 0.000} C_DIS
LIN {X -57.147,Y 28.575,Z -107.561,A 90.000,B 90.000,C 0.000} C_DIS
LIN {X -55.453,Y 28.575,Z -109.789,A 90.000,B 90.000,C 0.000} C_DIS
LIN {X -53.737,Y 28.575,Z -112.000,A 90.000,B 90.000,C 0.000} C_DIS
LIN {X -52.639,Y 28.575,Z -113.397,A 90.000,B 90.000,C 0.000} C_DIS
LIN {X -51.591,Y 28.575,Z -114.833,A 90.000,B 90.000,C 0.000} C_DIS
LIN {X -50.594,Y 28.575,Z -116.305,A 90.000,B 90.000,C 0.000} C_DIS
LIN {X -49.651,Y 28.575,Z -117.811,A 90.000,B 90.000,C 0.000} C_DIS
LIN {X -48.761,Y 28.575,Z -119.350,A 90.000,B 90.000,C 0.000} C_DIS
LIN {X -47.806,Y 28.575,Z -121.511,A 90.000,B 90.000,C 0.000} C_DIS
LIN {X -46.817,Y 28.575,Z -123.656,A 90.000,B 90.000,C 0.000} C_DIS
LIN {X -45.793,Y 28.575,Z -125.785,A 90.000,B 90.000,C 0.000} C_DIS
LIN {X -44.735,Y 28.575,Z -127.897,A 90.000,B 90.000,C 0.000} C_DIS
LIN {X -44.039,Y 28.575,Z -129.422,A 90.000,B 90.000,C 0.000} C_DIS
LIN {X -43.291,Y 28.575,Z -130.922,A 90.000,B 90.000,C 0.000} C_DIS
LIN {X -42.492,Y 28.575,Z -132.396,A 90.000,B 90.000,C 0.000} C_DIS
LIN {X -41.643,Y 28.575,Z -133.842,A 90.000,B 90.000,C 0.000} C_DIS
LIN {X -40.745,Y 28.575,Z -135.257,A 90.000,B 90.000,C 0.000} C_DIS
LIN {X -39.799,Y 28.575,Z -136.641,A 90.000,B 90.000,C 0.000} C_DIS
LIN {X -38.806,Y 28.575,Z -137.992,A 90.000,B 90.000,C 0.000} C_DIS
LIN {X -37.768,Y 28.575,Z -139.308,A 90.000,B 90.000,C 0.000} C_DIS
LIN {X -36.685,Y 28.575,Z -140.588,A 90.000,B 90.000,C 0.000} C_DIS
LIN {X -35.809,Y 28.575,Z -141.831,A 90.000,B 90.000,C 0.000} C_DIS
LIN {X -34.901,Y 28.575,Z -143.051,A 90.000,B 90.000,C 0.000} C_DIS
LIN {X -33.961,Y 28.575,Z -144.246,A 90.000,B 90.000,C 0.000} C_DIS
LIN {X -32.990,Y 28.575,Z -145.416,A 90.000,B 90.000,C 0.000} C_DIS
LIN {X -31.988,Y 28.575,Z -146.560,A 90.000,B 90.000,C 0.000} C_DIS
LIN {X -29.960,Y 28.575,Z -148.609,A 90.000,B 90.000,C 0.000} C_DIS
LIN {X -27.889,Y 28.575,Z -150.615,A 90.000,B 90.000,C 0.000} C_DIS
LIN {X -25.775,Y 28.575,Z -152.575,A 90.000,B 90.000,C 0.000} C_DIS
LIN {X -23.619,Y 28.575,Z -154.490,A 90.000,B 90.000,C 0.000} C_DIS
LIN {X -21.423,Y 28.575,Z -156.358,A 90.000,B 90.000,C 0.000} C_DIS
LIN {X -18.800,Y 28.575,Z -158.361,A 90.000,B 90.000,C 0.000} C_DIS
LIN {X -16.199,Y 28.575,Z -160.392,A 90.000,B 90.000,C 0.000} C_DIS
LIN {X -13.619,Y 28.575,Z -162.451,A 90.000,B 90.000,C 0.000} C_DIS
LIN {X -11.062,Y 28.575,Z -164.538,A 90.000,B 90.000,C 0.000} C_DIS
LIN {X -10.936,Y 28.575,Z -164.670,A 90.000,B 90.000,C 0.000} C_DIS
LIN {X -11.166,Y 28.575,Z -165.716,A 90.000,B 90.000,C 0.000} C_DIS
LIN {X -11.448,Y 28.575,Z -166.750,A 90.000,B 90.000,C 0.000} C_DIS
LIN {X -11.782,Y 28.575,Z -167.768,A 90.000,B 90.000,C 0.000} C_DIS
LIN {X -12.165,Y 28.575,Z -168.768,A 90.000,B 90.000,C 0.000} C_DIS
LIN {X -12.597,Y 28.575,Z -169.748,A 90.000,B 90.000,C 0.000} C_DIS
LIN {X -13.078,Y 28.575,Z -170.706,A 90.000,B 90.000,C 0.000} C_DIS
LIN {X -13.605,Y 28.575,Z -171.638,A 90.000,B 90.000,C 0.000} C_DIS
LIN {X -14.178,Y 28.575,Z -172.543,A 90.000,B 90.000,C 0.000} C_DIS
LIN {X -15.403,Y 28.575,Z -174.285,A 90.000,B 90.000,C 0.000} C_DIS
LIN {X -16.679,Y 28.575,Z -175.990,A 90.000,B 90.000,C 0.000} C_DIS
LIN {X -18.005,Y 28.575,Z -177.657,A 90.000,B 90.000,C 0.000} C_DIS
LIN {X -19.380,Y 28.575,Z -179.284,A 90.000,B 90.000,C 0.000} C_DIS
LIN {X -20.802,Y 28.575,Z -180.869,A 90.000,B 90.000,C 0.000} C_DIS
LIN {X -22.270,Y 28.575,Z -182.412,A 90.000,B 90.000,C 0.000} C_DIS
LIN {X -23.783,Y 28.575,Z -183.911,A 90.000,B 90.000,C 0.000} C_DIS
LIN {X -25.340,Y 28.575,Z -185.365,A 90.000,B 90.000,C 0.000} C_DIS
LIN {X -26.939,Y 28.575,Z -186.771,A 90.000,B 90.000,C 0.000} C_DIS
LIN {X -28.579,Y 28.575,Z -188.130,A 90.000,B 90.000,C 0.000} C_DIS
LIN {X -30.259,Y 28.575,Z -189.440,A 90.000,B 90.000,C 0.000} C_DIS
LIN {X -31.976,Y 28.575,Z -190.700,A 90.000,B 90.000,C 0.000} C_DIS
LIN {X -33.730,Y 28.575,Z -191.908,A 90.000,B 90.000,C 0.000} C_DIS
LIN {X -37.559,Y 28.575,Z -194.272,A 90.000,B 90.000,C 0.000} C_DIS
LIN {X -41.409,Y 28.575,Z -196.601,A 90.000,B 90.000,C 0.000} C_DIS
LIN {X -45.282,Y 28.575,Z -198.893,A 90.000,B 90.000,C 0.000} C_DIS
LIN {X -49.175,Y 28.575,Z -201.150,A 90.000,B 90.000,C 0.000} C_DIS
LIN {X -53.089,Y 28.575,Z -203.370,A 90.000,B 90.000,C 0.000} C_DIS
LIN {X -58.345,Y 28.575,Z -206.319,A 90.000,B 90.000,C 0.000} C_DIS
LIN {X -63.576,Y 28.575,Z -209.312,A 90.000,B 90.000,C 0.000} C_DIS
LIN {X -68.781,Y 28.575,Z -212.349,A 90.000,B 90.000,C 0.000} C_DIS
LIN {X -73.960,Y 28.575,Z -215.430,A 90.000,B 90.000,C 0.000} C_DIS
LIN {X -79.113,Y 28.575,Z -218.555,A 90.000,B 90.000,C 0.000} C_DIS
LIN {X -84.240,Y 28.575,Z -221.723,A 90.000,B 90.000,C 0.000} C_DIS
LIN {X -89.339,Y 28.575,Z -224.935,A 90.000,B 90.000,C 0.000} C_DIS
LIN {X -93.138,Y 28.575,Z -227.319,A 90.000,B 90.000,C 0.000} C_DIS
LIN {X -96.910,Y 28.575,Z -229.745,A 90.000,B 90.000,C 0.000} C_DIS
LIN {X -100.656,Y 28.575,Z -232.212,A 90.000,B 90.000,C 0.000} C_DIS
LIN {X -104.374,Y 28.575,Z -234.719,A 90.000,B 90.000,C 0.000} C_DIS
LIN {X -108.065,Y 28.575,Z -237.267,A 90.000,B 90.000,C 0.000} C_DIS
LIN {X -112.631,Y 28.575,Z -240.400,A 90.000,B 90.000,C 0.000} C_DIS
LIN {X -117.177,Y 28.575,Z -243.561,A 90.000,B 90.000,C 0.000} C_DIS
LIN {X -145.015,Y 28.575,Z -243.561,A 90.000,B 90.000,C 0.000} C_DIS
LIN {X -145.015,Y 28.575,Z 0.000,A 90.000,B 90.000,C 0.000} C_DIS
LIN {X 145.015,Y 28.575,Z 0.000,A 90.000,B 90.000,C 0.000} C_DIS
LIN {X 145.015,Y 28.575,Z -243.561,A 90.000,B 90.000,C 0.000} C_DIS
LIN {X 89.226,Y 28.575,Z -243.561,A 90.000,B 90.000,C 0.000} C_DIS
LIN {X 90.155,Y 28.575,Z -240.782,A 90.000,B 90.000,C 0.000} C_DIS
LIN {X 91.035,Y 28.575,Z -237.987,A 90.000,B 90.000,C 0.000} C_DIS
LIN {X 91.865,Y 28.575,Z -235.177,A 90.000,B 90.000,C 0.000} C_DIS
LIN {X 92.644,Y 28.575,Z -232.353,A 90.000,B 90.000,C 0.000} C_DIS
LIN {X 93.374,Y 28.575,Z -229.515,A 90.000,B 90.000,C 0.000} C_DIS
LIN {X 94.454,Y 28.575,Z -225.234,A 90.000,B 90.000,C 0.000} C_DIS
LIN {X 95.555,Y 28.575,Z -220.959,A 90.000,B 90.000,C 0.000} C_DIS
LIN {X 96.677,Y 28.575,Z -216.689,A 90.000,B 90.000,C 0.000} C_DIS
LIN {X 97.346,Y 28.575,Z -214.092,A 90.000,B 90.000,C 0.000} C_DIS
LIN {X 98.034,Y 28.575,Z -211.501,A 90.000,B 90.000,C 0.000} C_DIS
LIN {X 98.636,Y 28.575,Z -209.104,A 90.000,B 90.000,C 0.000} C_DIS
LIN {X 99.257,Y 28.575,Z -206.711,A 90.000,B 90.000,C 0.000} C_DIS
LIN {X 99.784,Y 28.575,Z -204.655,A 90.000,B 90.000,C 0.000} C_DIS
LIN {X 100.254,Y 28.575,Z -202.585,A 90.000,B 90.000,C 0.000} C_DIS
LIN {X 100.666,Y 28.575,Z -200.503,A 90.000,B 90.000,C 0.000} C_DIS
LIN {X 101.020,Y 28.575,Z -198.410,A 90.000,B 90.000,C 0.000} C_DIS
LIN {X 101.315,Y 28.575,Z -196.308,A 90.000,B 90.000,C 0.000} C_DIS
LIN {X 101.551,Y 28.575,Z -194.198,A 90.000,B 90.000,C 0.000} C_DIS
LIN {X 101.728,Y 28.575,Z -192.083,A 90.000,B 90.000,C 0.000} C_DIS
LIN {X 101.909,Y 28.575,Z -188.793,A 90.000,B 90.000,C 0.000} C_DIS
LIN {X 102.154,Y 28.575,Z -185.508,A 90.000,B 90.000,C 0.000} C_DIS
LIN {X 102.462,Y 28.575,Z -182.228,A 90.000,B 90.000,C 0.000} C_DIS
LIN {X 102.834,Y 28.575,Z -178.954,A 90.000,B 90.000,C 0.000} C_DIS
LIN {X 103.268,Y 28.575,Z -175.689,A 90.000,B 90.000,C 0.000} C_DIS
LIN {X 103.767,Y 28.575,Z -172.432,A 90.000,B 90.000,C 0.000} C_DIS
LIN {X 104.421,Y 28.575,Z -168.262,A 90.000,B 90.000,C 0.000} C_DIS
LIN {X 105.025,Y 28.575,Z -164.085,A 90.000,B 90.000,C 0.000} C_DIS
LIN {X 105.578,Y 28.575,Z -159.900,A 90.000,B 90.000,C 0.000} C_DIS
LIN {X 106.080,Y 28.575,Z -155.710,A 90.000,B 90.000,C 0.000} C_DIS
LIN {X 106.532,Y 28.575,Z -151.513,A 90.000,B 90.000,C 0.000} C_DIS
LIN {X 106.933,Y 28.575,Z -147.311,A 90.000,B 90.000,C 0.000} C_DIS
LIN {X 107.283,Y 28.575,Z -143.105,A 90.000,B 90.000,C 0.000} C_DIS
LIN {X 107.570,Y 28.575,Z -139.860,A 90.000,B 90.000,C 0.000} C_DIS
LIN {X 107.796,Y 28.575,Z -136.610,A 90.000,B 90.000,C 0.000} C_DIS
LIN {X 107.959,Y 28.575,Z -133.356,A 90.000,B 90.000,C 0.000} C_DIS
LIN {X 108.060,Y 28.575,Z -130.100,A 90.000,B 90.000,C 0.000} C_DIS
LIN {X 108.099,Y 28.575,Z -126.842,A 90.000,B 90.000,C 0.000} C_DIS
LIN {X 108.076,Y 28.575,Z -123.584,A 90.000,B 90.000,C 0.000} C_DIS
LIN {X 107.991,Y 28.575,Z -120.327,A 90.000,B 90.000,C 0.000} C_DIS
LIN {X 107.843,Y 28.575,Z -117.073,A 90.000,B 90.000,C 0.000} C_DIS
LIN {X 107.633,Y 28.575,Z -113.821,A 90.000,B 90.000,C 0.000} C_DIS
LIN {X 107.362,Y 28.575,Z -110.575,A 90.000,B 90.000,C 0.000} C_DIS
LIN {X 107.029,Y 28.575,Z -107.334,A 90.000,B 90.000,C 0.000} C_DIS
LIN {X 106.802,Y 28.575,Z -106.412,A 90.000,B 90.000,C 0.000} C_DIS
LIN {X 106.633,Y 28.575,Z -105.478,A 90.000,B 90.000,C 0.000} C_DIS
LIN {X 106.520,Y 28.575,Z -104.536,A 90.000,B 90.000,C 0.000} C_DIS
LIN {X 106.466,Y 28.575,Z -103.588,A 90.000,B 90.000,C 0.000} C_DIS
LIN {X 106.469,Y 28.575,Z -102.639,A 90.000,B 90.000,C 0.000} C_DIS
LIN {X 106.482,Y 28.575,Z -102.504,A 90.000,B 90.000,C 0.000} C_DIS
LIN {X 106.542,Y 28.575,Z -100.982,A 90.000,B 90.000,C 0.000} C_DIS
LIN {X 106.708,Y 28.575,Z -99.072,A 90.000,B 90.000,C 0.000} C_DIS
LIN {X 106.824,Y 28.575,Z -97.158,A 90.000,B 90.000,C 0.000} C_DIS
LIN {X 106.890,Y 28.575,Z -95.242,A 90.000,B 90.000,C 0.000} C_DIS
LIN {X 106.905,Y 28.575,Z -93.325,A 90.000,B 90.000,C 0.000} C_DIS
LIN {X 106.871,Y 28.575,Z -91.409,A 90.000,B 90.000,C 0.000} C_DIS
LIN {X 106.785,Y 28.575,Z -89.493,A 90.000,B 90.000,C 0.000} C_DIS
LIN {X 106.649,Y 28.575,Z -87.581,A 90.000,B 90.000,C 0.000} C_DIS
LIN {X 107.930,Y 28.575,Z -85.625,A 90.000,B 90.000,C 0.000} C_DIS
LIN {X 109.151,Y 28.575,Z -83.631,A 90.000,B 90.000,C 0.000} C_DIS
LIN {X 110.309,Y 28.575,Z -81.600,A 90.000,B 90.000,C 0.000} C_DIS
LIN {X 111.404,Y 28.575,Z -79.535,A 90.000,B 90.000,C 0.000} C_DIS
LIN {X 112.435,Y 28.575,Z -77.436,A 90.000,B 90.000,C 0.000} C_DIS
LIN {X 113.401,Y 28.575,Z -75.307,A 90.000,B 90.000,C 0.000} C_DIS
LIN {X 114.300,Y 28.575,Z -73.149,A 90.000,B 90.000,C 0.000} C_DIS
LIN {X 115.133,Y 28.575,Z -70.964,A 90.000,B 90.000,C 0.000} C_DIS
LIN {X 115.897,Y 28.575,Z -68.755,A 90.000,B 90.000,C 0.000} C_DIS
LIN {X 116.594,Y 28.575,Z -66.523,A 90.000,B 90.000,C 0.000} C_DIS
LIN {X 117.391,Y 28.575,Z -63.629,A 90.000,B 90.000,C 0.000} C_DIS
LIN {X 118.216,Y 28.575,Z -60.743,A 90.000,B 90.000,C 0.000} C_DIS
LIN {X 118.900,Y 28.575,Z -58.947,A 90.000,B 90.000,C 0.000} C_DIS
LIN {X 119.632,Y 28.575,Z -57.170,A 90.000,B 90.000,C 0.000} C_DIS
LIN {X 120.411,Y 28.575,Z -55.413,A 90.000,B 90.000,C 0.000} C_DIS
LIN {X 121.238,Y 28.575,Z -53.679,A 90.000,B 90.000,C 0.000} C_DIS
LIN {X 122.112,Y 28.575,Z -51.967,A 90.000,B 90.000,C 0.000} C_DIS
LIN {X 122.620,Y 28.575,Z -50.961,A 90.000,B 90.000,C 0.000} C_DIS
LIN {X 123.069,Y 28.575,Z -49.926,A 90.000,B 90.000,C 0.000} C_DIS
LIN {X 123.455,Y 28.575,Z -48.867,A 90.000,B 90.000,C 0.000} C_DIS
LIN {X 123.778,Y 28.575,Z -47.788,A 90.000,B 90.000,C 0.000} C_DIS
LIN {X 124.038,Y 28.575,Z -46.690,A 90.000,B 90.000,C 0.000} C_DIS
LIN {X 124.232,Y 28.575,Z -45.580,A 90.000,B 90.000,C 0.000} C_DIS
LIN {X 124.360,Y 28.575,Z -44.460,A 90.000,B 90.000,C 0.000} C_DIS
LIN {X 124.422,Y 28.575,Z -43.334,A 90.000,B 90.000,C 0.000} C_DIS
LIN {X 124.417,Y 28.575,Z -42.207,A 90.000,B 90.000,C 0.000} C_DIS
LIN {X 124.347,Y 28.575,Z -41.082,A 90.000,B 90.000,C 0.000} C_DIS
LIN {X 124.254,Y 28.575,Z -40.095,A 90.000,B 90.000,C 0.000} C_DIS
LIN {X 124.088,Y 28.575,Z -39.117,A 90.000,B 90.000,C 0.000} C_DIS
LIN {X 123.849,Y 28.575,Z -38.155,A 90.000,B 90.000,C 0.000} C_DIS
LIN {X 123.540,Y 28.575,Z -37.213,A 90.000,B 90.000,C 0.000} C_DIS
LIN {X 123.161,Y 28.575,Z -36.296,A 90.000,B 90.000,C 0.000} C_DIS
LIN {X 122.715,Y 28.575,Z -35.411,A 90.000,B 90.000,C 0.000} C_DIS
LIN {X 122.205,Y 28.575,Z -34.561,A 90.000,B 90.000,C 0.000} C_DIS
LIN {X 121.633,Y 28.575,Z -33.751,A 90.000,B 90.000,C 0.000} C_DIS
LIN {X 121.002,Y 28.575,Z -32.986,A 90.000,B 90.000,C 0.000} C_DIS
LIN {X 120.316,Y 28.575,Z -32.270,A 90.000,B 90.000,C 0.000} C_DIS
LIN {X 119.578,Y 28.575,Z -31.607,A 90.000,B 90.000,C 0.000} C_DIS
LIN {X 118.794,Y 28.575,Z -31.001,A 90.000,B 90.000,C 0.000} C_DIS
LIN {X 117.966,Y 28.575,Z -30.455,A 90.000,B 90.000,C 0.000} C_DIS
LIN {X 117.834,Y 28.575,Z -30.373,A 90.000,B 90.000,C 0.000} C_DIS
LIN {X 117.055,Y 28.575,Z -29.942,A 90.000,B 90.000,C 0.000} C_DIS
LIN {X 116.250,Y 28.575,Z -29.561,A 90.000,B 90.000,C 0.000} C_DIS
LIN {X 115.424,Y 28.575,Z -29.230,A 90.000,B 90.000,C 0.000} C_DIS
LIN {X 114.578,Y 28.575,Z -28.952,A 90.000,B 90.000,C 0.000} C_DIS
LIN {X 114.396,Y 28.575,Z -28.894,A 90.000,B 90.000,C 0.000} C_DIS
LIN {X 113.523,Y 28.575,Z -28.668,A 90.000,B 90.000,C 0.000} C_DIS
LIN {X 112.636,Y 28.575,Z -28.501,A 90.000,B 90.000,C 0.000} C_DIS
LIN {X 111.741,Y 28.575,Z -28.392,A 90.000,B 90.000,C 0.000} C_DIS
LIN {X 110.840,Y 28.575,Z -28.343,A 90.000,B 90.000,C 0.000} C_DIS
LIN {X 109.938,Y 28.575,Z -28.354,A 90.000,B 90.000,C 0.000} C_DIS
LIN {X 109.039,Y 28.575,Z -28.425,A 90.000,B 90.000,C 0.000} C_DIS
LIN {X 107.758,Y 28.575,Z -28.690,A 90.000,B 90.000,C 0.000} C_DIS
LIN {X 106.490,Y 28.575,Z -29.012,A 90.000,B 90.000,C 0.000} C_DIS
LIN {X 105.237,Y 28.575,Z -29.391,A 90.000,B 90.000,C 0.000} C_DIS
LIN {X 104.003,Y 28.575,Z -29.825,A 90.000,B 90.000,C 0.000} C_DIS
LIN {X 102.790,Y 28.575,Z -30.314,A 90.000,B 90.000,C 0.000} C_DIS
LIN {X 101.021,Y 28.575,Z -31.009,A 90.000,B 90.000,C 0.000} C_DIS
LIN {X 99.273,Y 28.575,Z -31.757,A 90.000,B 90.000,C 0.000} C_DIS
LIN {X 97.549,Y 28.575,Z -32.555,A 90.000,B 90.000,C 0.000} C_DIS
LIN {X 95.848,Y 28.575,Z -33.404,A 90.000,B 90.000,C 0.000} C_DIS
LIN {X 94.174,Y 28.575,Z -34.304,A 90.000,B 90.000,C 0.000} C_DIS
LIN {X 92.527,Y 28.575,Z -35.252,A 90.000,B 90.000,C 0.000} C_DIS
LIN {X 90.908,Y 28.575,Z -36.249,A 90.000,B 90.000,C 0.000} C_DIS
LIN {X 89.320,Y 28.575,Z -37.293,A 90.000,B 90.000,C 0.000} C_DIS
LIN {X 87.763,Y 28.575,Z -38.383,A 90.000,B 90.000,C 0.000} C_DIS
LIN {X 86.515,Y 28.575,Z -39.295,A 90.000,B 90.000,C 0.000} C_DIS
LIN {X 85.308,Y 28.575,Z -40.260,A 90.000,B 90.000,C 0.000} C_DIS
LIN {X 84.143,Y 28.575,Z -41.277,A 90.000,B 90.000,C 0.000} C_DIS
LIN {X 83.024,Y 28.575,Z -42.343,A 90.000,B 90.000,C 0.000} C_DIS
LIN {X 81.953,Y 28.575,Z -43.457,A 90.000,B 90.000,C 0.000} C_DIS
LIN {X 80.931,Y 28.575,Z -44.617,A 90.000,B 90.000,C 0.000} C_DIS
LIN {X 79.960,Y 28.575,Z -45.819,A 90.000,B 90.000,C 0.000} C_DIS
LIN {X 79.042,Y 28.575,Z -47.063,A 90.000,B 90.000,C 0.000} C_DIS
LIN {X 78.180,Y 28.575,Z -48.346,A 90.000,B 90.000,C 0.000} C_DIS
LIN {X 77.373,Y 28.575,Z -49.664,A 90.000,B 90.000,C 0.000} C_DIS
LIN {X 76.625,Y 28.575,Z -51.017,A 90.000,B 90.000,C 0.000} C_DIS
LIN {X 75.937,Y 28.575,Z -52.401,A 90.000,B 90.000,C 0.000} C_DIS
LIN {X 73.766,Y 28.575,Z -51.036,A 90.000,B 90.000,C 0.000} C_DIS
LIN {X 71.615,Y 28.575,Z -49.641,A 90.000,B 90.000,C 0.000} C_DIS
LIN {X 69.482,Y 28.575,Z -48.217,A 90.000,B 90.000,C 0.000} C_DIS
LIN {X 69.482,Y 41.075,Z -48.217,A 90.000,B 90.000,C 0.000} C_DIS
LIN {X 69.482,Y 53.575,Z -48.217,A 90.000,B 90.000,C 0.000} C_DIS
LIN {X 69.482,Y 54.814,Z -48.217,A 90.000,B 90.000,C 0.000} C_DIS
LIN {X -123.664,Y 54.814,Z -242.561,A 90.000,B 90.000,C 0.000} C_DIS
LIN {X -123.664,Y 46.431,Z -242.561,A 90.000,B 90.000,C 0.000} C_DIS
LIN {X -123.664,Y 33.931,Z -242.561,A 90.000,B 90.000,C 0.000} C_DIS
LIN {X -123.664,Y 21.431,Z -242.561,A 90.000,B 90.000,C 0.000} C_DIS
LIN {X -144.015,Y 21.431,Z -242.561,A 90.000,B 90.000,C 0.000} C_DIS
LIN {X -144.015,Y 21.431,Z -235.012,A 90.000,B 90.000,C 0.000} C_DIS
LIN {X -112.613,Y 21.431,Z -235.012,A 90.000,B 90.000,C 0.000} C_DIS
LIN {X -107.446,Y 21.431,Z -231.402,A 90.000,B 90.000,C 0.000} C_DIS
LIN {X -102.303,Y 21.431,Z -227.757,A 90.000,B 90.000,C 0.000} C_DIS
LIN {X -101.881,Y 21.431,Z -227.464,A 90.000,B 90.000,C 0.000} C_DIS
LIN {X -144.015,Y 21.431,Z -227.464,A 90.000,B 90.000,C 0.000} C_DIS
LIN {X -144.015,Y 21.431,Z -219.915,A 90.000,B 90.000,C 0.000} C_DIS
LIN {X -91.002,Y 21.431,Z -219.915,A 90.000,B 90.000,C 0.000} C_DIS
LIN {X -87.300,Y 21.431,Z -217.381,A 90.000,B 90.000,C 0.000} C_DIS
LIN {X -83.586,Y 21.431,Z -214.865,A 90.000,B 90.000,C 0.000} C_DIS
LIN {X -79.861,Y 21.431,Z -212.366,A 90.000,B 90.000,C 0.000} C_DIS
LIN {X -144.015,Y 21.431,Z -212.366,A 90.000,B 90.000,C 0.000} C_DIS
LIN {X -144.015,Y 21.431,Z -204.817,A 90.000,B 90.000,C 0.000} C_DIS
LIN {X -68.371,Y 21.431,Z -204.817,A 90.000,B 90.000,C 0.000} C_DIS
LIN {X -65.503,Y 21.431,Z -202.970,A 90.000,B 90.000,C 0.000} C_DIS
LIN {X -62.643,Y 21.431,Z -201.098,A 90.000,B 90.000,C 0.000} C_DIS
LIN {X -59.802,Y 21.431,Z -199.197,A 90.000,B 90.000,C 0.000} C_DIS
LIN {X -56.979,Y 21.431,Z -197.269,A 90.000,B 90.000,C 0.000} C_DIS
LIN {X -144.015,Y 21.431,Z -197.269,A 90.000,B 90.000,C 0.000} C_DIS
LIN {X -144.015,Y 21.431,Z -189.720,A 90.000,B 90.000,C 0.000} C_DIS
LIN {X -46.475,Y 21.431,Z -189.720,A 90.000,B 90.000,C 0.000} C_DIS
LIN {X -43.201,Y 21.431,Z -187.242,A 90.000,B 90.000,C 0.000} C_DIS
LIN {X -39.956,Y 21.431,Z -184.726,A 90.000,B 90.000,C 0.000} C_DIS
LIN {X -36.741,Y 21.431,Z -182.171,A 90.000,B 90.000,C 0.000} C_DIS
LIN {X -144.015,Y 21.431,Z -182.171,A 90.000,B 90.000,C 0.000} C_DIS
LIN {X -144.015,Y 21.431,Z -174.622,A 90.000,B 90.000,C 0.000} C_DIS
LIN {X -27.925,Y 21.431,Z -174.622,A 90.000,B 90.000,C 0.000} C_DIS
LIN {X -26.781,Y 21.431,Z -173.447,A 90.000,B 90.000,C 0.000} C_DIS
LIN {X -25.673,Y 21.431,Z -172.237,A 90.000,B 90.000,C 0.000} C_DIS
LIN {X -24.603,Y 21.431,Z -170.993,A 90.000,B 90.000,C 0.000} C_DIS
LIN {X -23.572,Y 21.431,Z -169.717,A 90.000,B 90.000,C 0.000} C_DIS
LIN {X -22.581,Y 21.431,Z -168.410,A 90.000,B 90.000,C 0.000} C_DIS
LIN {X -21.631,Y 21.431,Z -167.073,A 90.000,B 90.000,C 0.000} C_DIS
LIN {X -144.015,Y 21.431,Z -167.073,A 90.000,B 90.000,C 0.000} C_DIS
LIN {X -144.015,Y 21.431,Z -159.525,A 90.000,B 90.000,C 0.000} C_DIS
LIN {X -23.882,Y 21.431,Z -159.525,A 90.000,B 90.000,C 0.000} C_DIS
LIN {X -24.740,Y 21.431,Z -158.758,A 90.000,B 90.000,C 0.000} C_DIS
LIN {X -25.609,Y 21.431,Z -158.004,A 90.000,B 90.000,C 0.000} C_DIS
LIN {X -27.229,Y 21.431,Z -156.546,A 90.000,B 90.000,C 0.000} C_DIS
LIN {X -28.819,Y 21.431,Z -155.055,A 90.000,B 90.000,C 0.000} C_DIS
LIN {X -30.378,Y 21.431,Z -153.531,A 90.000,B 90.000,C 0.000} C_DIS
LIN {X -31.905,Y 21.431,Z -151.976,A 90.000,B 90.000,C 0.000} C_DIS
LIN {X -144.015,Y 21.431,Z -151.976,A 90.000,B 90.000,C 0.000} C_DIS
LIN {X -144.015,Y 21.431,Z -144.427,A 90.000,B 90.000,C 0.000} C_DIS
LIN {X -38.450,Y 21.431,Z -144.427,A 90.000,B 90.000,C 0.000} C_DIS
LIN {X -39.316,Y 21.431,Z -143.194,A 90.000,B 90.000,C 0.000} C_DIS
LIN {X -40.133,Y 21.431,Z -141.930,A 90.000,B 90.000,C 0.000} C_DIS
LIN {X -40.903,Y 21.431,Z -140.635,A 90.000,B 90.000,C 0.000} C_DIS
LIN {X -41.622,Y 21.431,Z -139.312,A 90.000,B 90.000,C 0.000} C_DIS
LIN {X -42.259,Y 21.431,Z -138.099,A 90.000,B 90.000,C 0.000} C_DIS
LIN {X -42.881,Y 21.431,Z -136.878,A 90.000,B 90.000,C 0.000} C_DIS
LIN {X -144.015,Y 21.431,Z -136.878,A 90.000,B 90.000,C 0.000} C_DIS
LIN {X -144.015,Y 21.431,Z -129.329,A 90.000,B 90.000,C 0.000} C_DIS
LIN {X -46.307,Y 21.431,Z -129.329,A 90.000,B 90.000,C 0.000} C_DIS
LIN {X -46.962,Y 21.431,Z -127.685,A 90.000,B 90.000,C 0.000} C_DIS
LIN {X -47.590,Y 21.431,Z -126.030,A 90.000,B 90.000,C 0.000} C_DIS
LIN {X -47.942,Y 21.431,Z -125.264,A 90.000,B 90.000,C 0.000} C_DIS
LIN {X -48.336,Y 21.431,Z -124.518,A 90.000,B 90.000,C 0.000} C_DIS
LIN {X -48.769,Y 21.431,Z -123.795,A 90.000,B 90.000,C 0.000} C_DIS
LIN {X -49.242,Y 21.431,Z -123.096,A 90.000,B 90.000,C 0.000} C_DIS
LIN {X -49.751,Y 21.431,Z -122.424,A 90.000,B 90.000,C 0.000} C_DIS
LIN {X -50.297,Y 21.431,Z -121.781,A 90.000,B 90.000,C 0.000} C_DIS
LIN {X -144.015,Y 21.431,Z -121.781,A 90.000,B 90.000,C 0.000} C_DIS
LIN {X -144.015,Y 21.431,Z -114.232,A 90.000,B 90.000,C 0.000} C_DIS
LIN {X -56.479,Y 21.431,Z -114.232,A 90.000,B 90.000,C 0.000} C_DIS
LIN {X -58.413,Y 21.431,Z -111.735,A 90.000,B 90.000,C 0.000} C_DIS
LIN {X -60.321,Y 21.431,Z -109.219,A 90.000,B 90.000,C 0.000} C_DIS
LIN {X -62.203,Y 21.431,Z -106.683,A 90.000,B 90.000,C 0.000} C_DIS
LIN {X -144.015,Y 21.431,Z -106.683,A 90.000,B 90.000,C 0.000} C_DIS
LIN {X -144.015,Y 21.431,Z -99.134,A 90.000,B 90.000,C 0.000} C_DIS
LIN {X -67.729,Y 21.431,Z -99.134,A 90.000,B 90.000,C 0.000} C_DIS
LIN {X -69.009,Y 21.431,Z -97.558,A 90.000,B 90.000,C 0.000} C_DIS
LIN {X -70.328,Y 21.431,Z -96.014,A 90.000,B 90.000,C 0.000} C_DIS
LIN {X -71.685,Y 21.431,Z -94.503,A 90.000,B 90.000,C 0.000} C_DIS
LIN {X -73.078,Y 21.431,Z -93.027,A 90.000,B 90.000,C 0.000} C_DIS
LIN {X -74.509,Y 21.431,Z -91.586,A 90.000,B 90.000,C 0.000} C_DIS
LIN {X -144.015,Y 21.431,Z -91.586,A 90.000,B 90.000,C 0.000} C_DIS
LIN {X -144.015,Y 21.431,Z -84.037,A 90.000,B 90.000,C 0.000} C_DIS
LIN {X -86.481,Y 21.431,Z -84.037,A 90.000,B 90.000,C 0.000} C_DIS
LIN {X -87.763,Y 21.431,Z -83.280,A 90.000,B 90.000,C 0.000} C_DIS
LIN {X -89.016,Y 21.431,Z -82.478,A 90.000,B 90.000,C 0.000} C_DIS
LIN {X -90.239,Y 21.431,Z -81.630,A 90.000,B 90.000,C 0.000} C_DIS
LIN {X -91.431,Y 21.431,Z -80.738,A 90.000,B 90.000,C 0.000} C_DIS
LIN {X -92.590,Y 21.431,Z -79.804,A 90.000,B 90.000,C 0.000} C_DIS
LIN {X -93.714,Y 21.431,Z -78.829,A 90.000,B 90.000,C 0.000} C_DIS
LIN {X -94.348,Y 21.431,Z -78.307,A 90.000,B 90.000,C 0.000} C_DIS
LIN {X -94.973,Y 21.431,Z -77.775,A 90.000,B 90.000,C 0.000} C_DIS
LIN {X -95.097,Y 21.431,Z -77.681,A 90.000,B 90.000,C 0.000} C_DIS
LIN {X -95.407,Y 21.431,Z -77.405,A 90.000,B 90.000,C 0.000} C_DIS
LIN {X -95.742,Y 21.431,Z -77.160,A 90.000,B 90.000,C 0.000} C_DIS
LIN {X -95.872,Y 21.431,Z -77.087,A 90.000,B 90.000,C 0.000} C_DIS
LIN {X -96.814,Y 21.431,Z -76.488,A 90.000,B 90.000,C 0.000} C_DIS
LIN {X -144.015,Y 21.431,Z -76.488,A 90.000,B 90.000,C 0.000} C_DIS
LIN {X -144.015,Y 21.431,Z -68.939,A 90.000,B 90.000,C 0.000} C_DIS
LIN {X -107.000,Y 21.431,Z -68.939,A 90.000,B 90.000,C 0.000} C_DIS
LIN {X -108.476,Y 21.431,Z -67.541,A 90.000,B 90.000,C 0.000} C_DIS
LIN {X -109.906,Y 21.431,Z -66.097,A 90.000,B 90.000,C 0.000} C_DIS
LIN {X -111.290,Y 21.431,Z -64.609,A 90.000,B 90.000,C 0.000} C_DIS
LIN {X -112.627,Y 21.431,Z -63.077,A 90.000,B 90.000,C 0.000} C_DIS
LIN {X -113.914,Y 21.431,Z -61.504,A 90.000,B 90.000,C 0.000} C_DIS
LIN {X -113.997,Y 21.431,Z -61.390,A 90.000,B 90.000,C 0.000} C_DIS
LIN {X -144.015,Y 21.431,Z -61.390,A 90.000,B 90.000,C 0.000} C_DIS
LIN {X -144.015,Y 21.431,Z -53.842,A 90.000,B 90.000,C 0.000} C_DIS
LIN {X -117.257,Y 21.431,Z -53.842,A 90.000,B 90.000,C 0.000} C_DIS
LIN {X -117.409,Y 21.431,Z -52.919,A 90.000,B 90.000,C 0.000} C_DIS
LIN {X -117.514,Y 21.431,Z -51.989,A 90.000,B 90.000,C 0.000} C_DIS
LIN {X -117.574,Y 21.431,Z -51.055,A 90.000,B 90.000,C 0.000} C_DIS
LIN {X -117.587,Y 21.431,Z -50.120,A 90.000,B 90.000,C 0.000} C_DIS
LIN {X -117.553,Y 21.431,Z -49.185,A 90.000,B 90.000,C 0.000} C_DIS
LIN {X -117.497,Y 21.431,Z -48.722,A 90.000,B 90.000,C 0.000} C_DIS
LIN {X -117.414,Y 21.431,Z -48.264,A 90.000,B 90.000,C 0.000} C_DIS
LIN {X -117.647,Y 21.431,Z -47.616,A 90.000,B 90.000,C 0.000} C_DIS
LIN {X -117.854,Y 21.431,Z -46.958,A 90.000,B 90.000,C 0.000} C_DIS
LIN {X -118.034,Y 21.431,Z -46.293,A 90.000,B 90.000,C 0.000} C_DIS
LIN {X -144.015,Y 21.431,Z -46.293,A 90.000,B 90.000,C 0.000} C_DIS
LIN {X -144.015,Y 21.431,Z -38.744,A 90.000,B 90.000,C 0.000} C_DIS
LIN {X -118.185,Y 21.431,Z -38.744,A 90.000,B 90.000,C 0.000} C_DIS
LIN {X -118.018,Y 21.431,Z -38.016,A 90.000,B 90.000,C 0.000} C_DIS
LIN {X -117.819,Y 21.431,Z -37.297,A 90.000,B 90.000,C 0.000} C_DIS
LIN {X -117.589,Y 21.431,Z -36.587,A 90.000,B 90.000,C 0.000} C_DIS
LIN {X -117.328,Y 21.431,Z -35.887,A 90.000,B 90.000,C 0.000} C_DIS
LIN {X -116.548,Y 21.431,Z -34.383,A 90.000,B 90.000,C 0.000} C_DIS
LIN {X -116.453,Y 21.431,Z -34.233,A 90.000,B 90.000,C 0.000} C_DIS
LIN {X -115.976,Y 21.431,Z -33.508,A 90.000,B 90.000,C 0.000} C_DIS
LIN {X -115.450,Y 21.431,Z -32.817,A 90.000,B 90.000,C 0.000} C_DIS
LIN {X -114.879,Y 21.431,Z -32.163,A 90.000,B 90.000,C 0.000} C_DIS
LIN {X -114.265,Y 21.431,Z -31.549,A 90.000,B 90.000,C 0.000} C_DIS
LIN {X -114.105,Y 21.431,Z -31.401,A 90.000,B 90.000,C 0.000} C_DIS
LIN {X -113.852,Y 21.431,Z -31.195,A 90.000,B 90.000,C 0.000} C_DIS
LIN {X -144.015,Y 21.431,Z -31.195,A 90.000,B 90.000,C 0.000} C_DIS
LIN {X -144.015,Y 21.431,Z -23.646,A 90.000,B 90.000,C 0.000} C_DIS
LIN {X -104.728,Y 21.431,Z -23.646,A 90.000,B 90.000,C 0.000} C_DIS
LIN {X -104.135,Y 21.431,Z -22.834,A 90.000,B 90.000,C 0.000} C_DIS
LIN {X -103.497,Y 21.431,Z -22.057,A 90.000,B 90.000,C 0.000} C_DIS
LIN {X -102.816,Y 21.431,Z -21.317,A 90.000,B 90.000,C 0.000} C_DIS
LIN {X -102.095,Y 21.431,Z -20.616,A 90.000,B 90.000,C 0.000} C_DIS
LIN {X -101.336,Y 21.431,Z -19.957,A 90.000,B 90.000,C 0.000} C_DIS
LIN {X -100.541,Y 21.431,Z -19.342,A 90.000,B 90.000,C 0.000} C_DIS
LIN {X -100.370,Y 21.431,Z -19.225,A 90.000,B 90.000,C 0.000} C_DIS
LIN {X -99.688,Y 21.431,Z -18.780,A 90.000,B 90.000,C 0.000} C_DIS
LIN {X -98.976,Y 21.431,Z -18.384,A 90.000,B 90.000,C 0.000} C_DIS
LIN {X -98.239,Y 21.431,Z -18.038,A 90.000,B 90.000,C 0.000} C_DIS
LIN {X -97.479,Y 21.431,Z -17.744,A 90.000,B 90.000,C 0.000} C_DIS
LIN {X -97.327,Y 21.431,Z -17.689,A 90.000,B 90.000,C 0.000} C_DIS
LIN {X -96.487,Y 21.431,Z -17.435,A 90.000,B 90.000,C 0.000} C_DIS
LIN {X -95.635,Y 21.431,Z -17.229,A 90.000,B 90.000,C 0.000} C_DIS
LIN {X -94.772,Y 21.431,Z -17.071,A 90.000,B 90.000,C 0.000} C_DIS
LIN {X -93.901,Y 21.431,Z -16.962,A 90.000,B 90.000,C 0.000} C_DIS
LIN {X -93.026,Y 21.431,Z -16.903,A 90.000,B 90.000,C 0.000} C_DIS
LIN {X -92.149,Y 21.431,Z -16.894,A 90.000,B 90.000,C 0.000} C_DIS
LIN {X -91.979,Y 21.431,Z -16.493,A 90.000,B 90.000,C 0.000} C_DIS
LIN {X -91.796,Y 21.431,Z -16.098,A 90.000,B 90.000,C 0.000} C_DIS
LIN {X -144.015,Y 21.431,Z -16.098,A 90.000,B 90.000,C 0.000} C_DIS
LIN {X -144.015,Y 21.431,Z -8.549,A 90.000,B 90.000,C 0.000} C_DIS
LIN {X -81.686,Y 21.431,Z -8.549,A 90.000,B 90.000,C 0.000} C_DIS
LIN {X -80.686,Y 21.431,Z -8.361,A 90.000,B 90.000,C 0.000} C_DIS
LIN {X -79.677,Y 21.431,Z -8.235,A 90.000,B 90.000,C 0.000} C_DIS
LIN {X -78.662,Y 21.431,Z -8.172,A 90.000,B 90.000,C 0.000} C_DIS
LIN {X -77.644,Y 21.431,Z -8.172,A 90.000,B 90.000,C 0.000} C_DIS
LIN {X -76.629,Y 21.431,Z -8.235,A 90.000,B 90.000,C 0.000} C_DIS
LIN {X -75.620,Y 21.431,Z -8.361,A 90.000,B 90.000,C 0.000} C_DIS
LIN {X -74.620,Y 21.431,Z -8.549,A 90.000,B 90.000,C 0.000} C_DIS
LIN {X 144.015,Y 21.431,Z -8.549,A 90.000,B 90.000,C 0.000} C_DIS
LIN {X 144.015,Y 21.431,Z -16.098,A 90.000,B 90.000,C 0.000} C_DIS
LIN {X -61.432,Y 21.431,Z -16.098,A 90.000,B 90.000,C 0.000} C_DIS
LIN {X -60.630,Y 21.431,Z -16.954,A 90.000,B 90.000,C 0.000} C_DIS
LIN {X -59.865,Y 21.431,Z -17.844,A 90.000,B 90.000,C 0.000} C_DIS
LIN {X -59.139,Y 21.431,Z -18.765,A 90.000,B 90.000,C 0.000} C_DIS
LIN {X -58.452,Y 21.431,Z -19.716,A 90.000,B 90.000,C 0.000} C_DIS
LIN {X -57.962,Y 21.431,Z -20.600,A 90.000,B 90.000,C 0.000} C_DIS
LIN {X -57.497,Y 21.431,Z -21.498,A 90.000,B 90.000,C 0.000} C_DIS
LIN {X -57.058,Y 21.431,Z -22.409,A 90.000,B 90.000,C 0.000} C_DIS
LIN {X -55.818,Y 21.431,Z -22.761,A 90.000,B 90.000,C 0.000} C_DIS
LIN {X -54.565,Y 21.431,Z -23.061,A 90.000,B 90.000,C 0.000} C_DIS
LIN {X -53.300,Y 21.431,Z -23.309,A 90.000,B 90.000,C 0.000} C_DIS
LIN {X -52.026,Y 21.431,Z -23.504,A 90.000,B 90.000,C 0.000} C_DIS
LIN {X -50.745,Y 21.431,Z -23.646,A 90.000,B 90.000,C 0.000} C_DIS
LIN {X 144.015,Y 21.431,Z -23.646,A 90.000,B 90.000,C 0.000} C_DIS
LIN {X 144.015,Y 21.431,Z -31.195,A 90.000,B 90.000,C 0.000} C_DIS
LIN {X 120.629,Y 21.431,Z -31.195,A 90.000,B 90.000,C 0.000} C_DIS
LIN {X 121.339,Y 21.431,Z -31.880,A 90.000,B 90.000,C 0.000} C_DIS
LIN {X 122.000,Y 21.431,Z -32.612,A 90.000,B 90.000,C 0.000} C_DIS
LIN {X 122.609,Y 21.431,Z -33.388,A 90.000,B 90.000,C 0.000} C_DIS
LIN {X 123.163,Y 21.431,Z -34.204,A 90.000,B 90.000,C 0.000} C_DIS
LIN {X 123.660,Y 21.431,Z -35.056,A 90.000,B 90.000,C 0.000} C_DIS
LIN {X 124.097,Y 21.431,Z -35.941,A 90.000,B 90.000,C 0.000} C_DIS
LIN {X 124.472,Y 21.431,Z -36.853,A 90.000,B 90.000,C 0.000} C_DIS
LIN {X 124.783,Y 21.431,Z -37.789,A 90.000,B 90.000,C 0.000} C_DIS
LIN {X 125.030,Y 21.431,Z -38.744,A 90.000,B 90.000,C 0.000} C_DIS
LIN {X 144.015,Y 21.431,Z -38.744,A 90.000,B 90.000,C 0.000} C_DIS
LIN {X 144.015,Y 21.431,Z -46.293,A 90.000,B 90.000,C 0.000} C_DIS
LIN {X 125.131,Y 21.431,Z -46.293,A 90.000,B 90.000,C 0.000} C_DIS
LIN {X 124.915,Y 21.431,Z -47.361,A 90.000,B 90.000,C 0.000} C_DIS
LIN {X 124.642,Y 21.431,Z -48.415,A 90.000,B 90.000,C 0.000} C_DIS
LIN {X 124.313,Y 21.431,Z -49.453,A 90.000,B 90.000,C 0.000} C_DIS
LIN {X 123.927,Y 21.431,Z -50.472,A 90.000,B 90.000,C 0.000} C_DIS
LIN {X 123.487,Y 21.431,Z -51.468,A 90.000,B 90.000,C 0.000} C_DIS
LIN {X 122.993,Y 21.431,Z -52.439,A 90.000,B 90.000,C 0.000} C_DIS
LIN {X 122.629,Y 21.431,Z -53.138,A 90.000,B 90.000,C 0.000} C_DIS
LIN {X 122.274,Y 21.431,Z -53.842,A 90.000,B 90.000,C 0.000} C_DIS
LIN {X 144.015,Y 21.431,Z -53.842,A 90.000,B 90.000,C 0.000} C_DIS
LIN {X 144.015,Y 21.431,Z -61.390,A 90.000,B 90.000,C 0.000} C_DIS
LIN {X 119.069,Y 21.431,Z -61.390,A 90.000,B 90.000,C 0.000} C_DIS
LIN {X 118.300,Y 21.431,Z -64.088,A 90.000,B 90.000,C 0.000} C_DIS
LIN {X 117.556,Y 21.431,Z -66.794,A 90.000,B 90.000,C 0.000} C_DIS
LIN {X 117.230,Y 21.431,Z -67.869,A 90.000,B 90.000,C 0.000} C_DIS
LIN {X 116.890,Y 21.431,Z -68.939,A 90.000,B 90.000,C 0.000} C_DIS
LIN {X 144.015,Y 21.431,Z -68.939,A 90.000,B 90.000,C 0.000} C_DIS
LIN {X 144.015,Y 21.431,Z -76.488,A 90.000,B 90.000,C 0.000} C_DIS
LIN {X 113.973,Y 21.431,Z -76.488,A 90.000,B 90.000,C 0.000} C_DIS
LIN {X 113.077,Y 21.431,Z -78.415,A 90.000,B 90.000,C 0.000} C_DIS
LIN {X 112.128,Y 21.431,Z -80.317,A 90.000,B 90.000,C 0.000} C_DIS
LIN {X 111.126,Y 21.431,Z -82.191,A 90.000,B 90.000,C 0.000} C_DIS
LIN {X 110.073,Y 21.431,Z -84.037,A 90.000,B 90.000,C 0.000} C_DIS
LIN {X 144.015,Y 21.431,Z -84.037,A 90.000,B 90.000,C 0.000} C_DIS
LIN {X 144.015,Y 21.431,Z -91.586,A 90.000,B 90.000,C 0.000} C_DIS
LIN {X 108.647,Y 21.431,Z -91.586,A 90.000,B 90.000,C 0.000} C_DIS
LIN {X 108.961,Y 21.431,Z -93.137,A 90.000,B 90.000,C 0.000} C_DIS
LIN {X 109.237,Y 21.431,Z -94.696,A 90.000,B 90.000,C 0.000} C_DIS
LIN {X 109.474,Y 21.431,Z -96.261,A 90.000,B 90.000,C 0.000} C_DIS
LIN {X 109.672,Y 21.431,Z -97.832,A 90.000,B 90.000,C 0.000} C_DIS
LIN {X 109.677,Y 21.431,Z -97.906,A 90.000,B 90.000,C 0.000} C_DIS
LIN {X 109.864,Y 21.431,Z -99.134,A 90.000,B 90.000,C 0.000} C_DIS
LIN {X 144.015,Y 21.431,Z -99.134,A 90.000,B 90.000,C 0.000} C_DIS
LIN {X 144.015,Y 21.431,Z -106.683,A 90.000,B 90.000,C 0.000} C_DIS
LIN {X 110.968,Y 21.431,Z -106.683,A 90.000,B 90.000,C 0.000} C_DIS
LIN {X 111.464,Y 21.431,Z -110.455,A 90.000,B 90.000,C 0.000} C_DIS
LIN {X 111.920,Y 21.431,Z -114.232,A 90.000,B 90.000,C 0.000} C_DIS
LIN {X 144.015,Y 21.431,Z -114.232,A 90.000,B 90.000,C 0.000} C_DIS
LIN {X 144.015,Y 21.431,Z -121.781,A 90.000,B 90.000,C 0.000} C_DIS
LIN {X 112.708,Y 21.431,Z -121.781,A 90.000,B 90.000,C 0.000} C_DIS
LIN {X 112.891,Y 21.431,Z -123.802,A 90.000,B 90.000,C 0.000} C_DIS
LIN {X 113.064,Y 21.431,Z -125.824,A 90.000,B 90.000,C 0.000} C_DIS
LIN {X 113.147,Y 21.431,Z -127.576,A 90.000,B 90.000,C 0.000} C_DIS
LIN {X 113.211,Y 21.431,Z -129.329,A 90.000,B 90.000,C 0.000} C_DIS
LIN {X 144.015,Y 21.431,Z -129.329,A 90.000,B 90.000,C 0.000} C_DIS
LIN {X 144.015,Y 21.431,Z -136.878,A 90.000,B 90.000,C 0.000} C_DIS
LIN {X 113.282,Y 21.431,Z -136.878,A 90.000,B 90.000,C 0.000} C_DIS
LIN {X 113.231,Y 21.431,Z -139.396,A 90.000,B 90.000,C 0.000} C_DIS
LIN {X 113.142,Y 21.431,Z -141.912,A 90.000,B 90.000,C 0.000} C_DIS
LIN {X 113.015,Y 21.431,Z -144.427,A 90.000,B 90.000,C 0.000} C_DIS
LIN {X 144.015,Y 21.431,Z -144.427,A 90.000,B 90.000,C 0.000} C_DIS
LIN {X 144.015,Y 21.431,Z -151.976,A 90.000,B 90.000,C 0.000} C_DIS
LIN {X 112.456,Y 21.431,Z -151.976,A 90.000,B 90.000,C 0.000} C_DIS
LIN {X 112.157,Y 21.431,Z -155.752,A 90.000,B 90.000,C 0.000} C_DIS
LIN {X 111.830,Y 21.431,Z -159.525,A 90.000,B 90.000,C 0.000} C_DIS
LIN {X 144.015,Y 21.431,Z -159.525,A 90.000,B 90.000,C 0.000} C_DIS
LIN {X 144.015,Y 21.431,Z -167.073,A 90.000,B 90.000,C 0.000} C_DIS
LIN {X 111.095,Y 21.431,Z -167.073,A 90.000,B 90.000,C 0.000} C_DIS
LIN {X 110.686,Y 21.431,Z -170.849,A 90.000,B 90.000,C 0.000} C_DIS
LIN {X 110.250,Y 21.431,Z -174.622,A 90.000,B 90.000,C 0.000} C_DIS
LIN {X 144.015,Y 21.431,Z -174.622,A 90.000,B 90.000,C 0.000} C_DIS
LIN {X 144.015,Y 21.431,Z -182.171,A 90.000,B 90.000,C 0.000} C_DIS
LIN {X 109.294,Y 21.431,Z -182.171,A 90.000,B 90.000,C 0.000} C_DIS
LIN {X 108.774,Y 21.431,Z -185.947,A 90.000,B 90.000,C 0.000} C_DIS
LIN {X 108.227,Y 21.431,Z -189.720,A 90.000,B 90.000,C 0.000} C_DIS
LIN {X 144.015,Y 21.431,Z -189.720,A 90.000,B 90.000,C 0.000} C_DIS
LIN {X 144.015,Y 21.431,Z -197.269,A 90.000,B 90.000,C 0.000} C_DIS
LIN {X 107.016,Y 21.431,Z -197.269,A 90.000,B 90.000,C 0.000} C_DIS
LIN {X 106.566,Y 21.431,Z -199.789,A 90.000,B 90.000,C 0.000} C_DIS
LIN {X 106.092,Y 21.431,Z -202.305,A 90.000,B 90.000,C 0.000} C_DIS
LIN {X 105.597,Y 21.431,Z -204.817,A 90.000,B 90.000,C 0.000} C_DIS
LIN {X 144.015,Y 21.431,Z -204.817,A 90.000,B 90.000,C 0.000} C_DIS
LIN {X 144.015,Y 21.431,Z -212.366,A 90.000,B 90.000,C 0.000} C_DIS
LIN {X 103.963,Y 21.431,Z -212.366,A 90.000,B 90.000,C 0.000} C_DIS
LIN {X 103.369,Y 21.431,Z -214.888,A 90.000,B 90.000,C 0.000} C_DIS
LIN {X 102.752,Y 21.431,Z -217.404,A 90.000,B 90.000,C 0.000} C_DIS
LIN {X 102.112,Y 21.431,Z -219.915,A 90.000,B 90.000,C 0.000} C_DIS
LIN {X 144.015,Y 21.431,Z -219.915,A 90.000,B 90.000,C 0.000} C_DIS
LIN {X 144.015,Y 21.431,Z -227.464,A 90.000,B 90.000,C 0.000} C_DIS
LIN {X 100.174,Y 21.431,Z -227.464,A 90.000,B 90.000,C 0.000} C_DIS
LIN {X 99.489,Y 21.431,Z -229.986,A 90.000,B 90.000,C 0.000} C_DIS
LIN {X 98.785,Y 21.431,Z -232.502,A 90.000,B 90.000,C 0.000} C_DIS
LIN {X 98.060,Y 21.431,Z -235.012,A 90.000,B 90.000,C 0.000} C_DIS
LIN {X 144.015,Y 21.431,Z -235.012,A 90.000,B 90.000,C 0.000} C_DIS
LIN {X 144.015,Y 21.431,Z -242.561,A 90.000,B 90.000,C 0.000} C_DIS
LIN {X 95.750,Y 21.431,Z -242.561,A 90.000,B 90.000,C 0.000} C_DIS
LIN {X 97.098,Y 21.431,Z -238.236,A 90.000,B 90.000,C 0.000} C_DIS
LIN {X 98.386,Y 21.431,Z -233.893,A 90.000,B 90.000,C 0.000} C_DIS
LIN {X 99.614,Y 21.431,Z -229.533,A 90.000,B 90.000,C 0.000} C_DIS
LIN {X 100.782,Y 21.431,Z -225.156,A 90.000,B 90.000,C 0.000} C_DIS
LIN {X 101.890,Y 21.431,Z -220.764,A 90.000,B 90.000,C 0.000} C_DIS
LIN {X 102.852,Y 21.431,Z -217.004,A 90.000,B 90.000,C 0.000} C_DIS
LIN {X 103.762,Y 21.431,Z -213.232,A 90.000,B 90.000,C 0.000} C_DIS
LIN {X 104.620,Y 21.431,Z -209.448,A 90.000,B 90.000,C 0.000} C_DIS
LIN {X 105.427,Y 21.431,Z -205.652,A 90.000,B 90.000,C 0.000} C_DIS
LIN {X 106.181,Y 21.431,Z -201.845,A 90.000,B 90.000,C 0.000} C_DIS
LIN {X 106.883,Y 21.431,Z -198.028,A 90.000,B 90.000,C 0.000} C_DIS
LIN {X 107.533,Y 21.431,Z -194.202,A 90.000,B 90.000,C 0.000} C_DIS
LIN {X 108.130,Y 21.431,Z -190.368,A 90.000,B 90.000,C 0.000} C_DIS
LIN {X 108.961,Y 21.431,Z -184.615,A 90.000,B 90.000,C 0.000} C_DIS
LIN {X 109.728,Y 21.431,Z -178.853,A 90.000,B 90.000,C 0.000} C_DIS
LIN {X 110.431,Y 21.431,Z -173.083,A 90.000,B 90.000,C 0.000} C_DIS
LIN {X 111.071,Y 21.431,Z -167.306,A 90.000,B 90.000,C 0.000} C_DIS
LIN {X 111.647,Y 21.431,Z -161.522,A 90.000,B 90.000,C 0.000} C_DIS
LIN {X 112.159,Y 21.431,Z -155.731,A 90.000,B 90.000,C 0.000} C_DIS
LIN {X 112.606,Y 21.431,Z -149.936,A 90.000,B 90.000,C 0.000} C_DIS
LIN {X 112.851,Y 21.431,Z -146.929,A 90.000,B 90.000,C 0.000} C_DIS
LIN {X 113.043,Y 21.431,Z -143.918,A 90.000,B 90.000,C 0.000} C_DIS
LIN {X 113.181,Y 21.431,Z -140.904,A 90.000,B 90.000,C 0.000} C_DIS
LIN {X 113.265,Y 21.431,Z -137.888,A 90.000,B 90.000,C 0.000} C_DIS
LIN {X 113.295,Y 21.431,Z -134.871,A 90.000,B 90.000,C 0.000} C_DIS
LIN {X 113.272,Y 21.431,Z -131.854,A 90.000,B 90.000,C 0.000} C_DIS
LIN {X 113.194,Y 21.431,Z -128.838,A 90.000,B 90.000,C 0.000} C_DIS
LIN {X 113.064,Y 21.431,Z -125.824,A 90.000,B 90.000,C 0.000} C_DIS
LIN {X 112.672,Y 21.431,Z -121.393,A 90.000,B 90.000,C 0.000} C_DIS
LIN {X 112.225,Y 21.431,Z -116.966,A 90.000,B 90.000,C 0.000} C_DIS
LIN {X 111.722,Y 21.431,Z -112.546,A 90.000,B 90.000,C 0.000} C_DIS
LIN {X 111.163,Y 21.431,Z -108.132,A 90.000,B 90.000,C 0.000} C_DIS
LIN {X 110.550,Y 21.431,Z -103.726,A 90.000,B 90.000,C 0.000} C_DIS
LIN {X 109.881,Y 21.431,Z -99.328,A 90.000,B 90.000,C 0.000} C_DIS
LIN {X 109.866,Y 21.431,Z -99.146,A 90.000,B 90.000,C 0.000} C_DIS
LIN {X 109.677,Y 21.431,Z -97.906,A 90.000,B 90.000,C 0.000} C_DIS
LIN {X 109.672,Y 21.431,Z -97.832,A 90.000,B 90.000,C 0.000} C_DIS
LIN {X 109.420,Y 21.431,Z -95.881,A 90.000,B 90.000,C 0.000} C_DIS
LIN {X 109.108,Y 21.431,Z -93.938,A 90.000,B 90.000,C 0.000} C_DIS
LIN {X 108.737,Y 21.431,Z -92.006,A 90.000,B 90.000,C 0.000} C_DIS
LIN {X 108.305,Y 21.431,Z -90.087,A 90.000,B 90.000,C 0.000} C_DIS
LIN {X 108.095,Y 21.431,Z -89.672,A 90.000,B 90.000,C 0.000} C_DIS
LIN {X 107.924,Y 21.431,Z -89.240,A 90.000,B 90.000,C 0.000} C_DIS
LIN {X 107.794,Y 21.431,Z -88.794,A 90.000,B 90.000,C 0.000} C_DIS
LIN {X 107.704,Y 21.431,Z -88.337,A 90.000,B 90.000,C 0.000} C_DIS
LIN {X 107.657,Y 21.431,Z -87.875,A 90.000,B 90.000,C 0.000} C_DIS
LIN {X 108.931,Y 21.431,Z -85.914,A 90.000,B 90.000,C 0.000} C_DIS
LIN {X 110.144,Y 21.431,Z -83.916,A 90.000,B 90.000,C 0.000} C_DIS
LIN {X 111.296,Y 21.431,Z -81.882,A 90.000,B 90.000,C 0.000} C_DIS
LIN {X 112.385,Y 21.431,Z -79.813,A 90.000,B 90.000,C 0.000} C_DIS
LIN {X 113.411,Y 21.431,Z -77.712,A 90.000,B 90.000,C 0.000} C_DIS
LIN {X 114.372,Y 21.431,Z -75.581,A 90.000,B 90.000,C 0.000} C_DIS
LIN {X 115.268,Y 21.431,Z -73.422,A 90.000,B 90.000,C 0.000} C_DIS
LIN {X 116.098,Y 21.431,Z -71.236,A 90.000,B 90.000,C 0.000} C_DIS
LIN {X 116.861,Y 21.431,Z -69.026,A 90.000,B 90.000,C 0.000} C_DIS
LIN {X 117.556,Y 21.431,Z -66.794,A 90.000,B 90.000,C 0.000} C_DIS
LIN {X 118.347,Y 21.431,Z -63.920,A 90.000,B 90.000,C 0.000} C_DIS
LIN {X 119.167,Y 21.431,Z -61.055,A 90.000,B 90.000,C 0.000} C_DIS
LIN {X 119.839,Y 21.431,Z -59.292,A 90.000,B 90.000,C 0.000} C_DIS
LIN {X 120.558,Y 21.431,Z -57.547,A 90.000,B 90.000,C 0.000} C_DIS
LIN {X 121.324,Y 21.431,Z -55.823,A 90.000,B 90.000,C 0.000} C_DIS
LIN {X 122.136,Y 21.431,Z -54.120,A 90.000,B 90.000,C 0.000} C_DIS
LIN {X 122.993,Y 21.431,Z -52.439,A 90.000,B 90.000,C 0.000} C_DIS
LIN {X 123.527,Y 21.431,Z -51.382,A 90.000,B 90.000,C 0.000} C_DIS
LIN {X 123.997,Y 21.431,Z -50.296,A 90.000,B 90.000,C 0.000} C_DIS
LIN {X 124.403,Y 21.431,Z -49.184,A 90.000,B 90.000,C 0.000} C_DIS
LIN {X 124.743,Y 21.431,Z -48.050,A 90.000,B 90.000,C 0.000} C_DIS
LIN {X 125.015,Y 21.431,Z -46.898,A 90.000,B 90.000,C 0.000} C_DIS
LIN {X 125.220,Y 21.431,Z -45.732,A 90.000,B 90.000,C 0.000} C_DIS
LIN {X 125.355,Y 21.431,Z -44.556,A 90.000,B 90.000,C 0.000} C_DIS
LIN {X 125.421,Y 21.431,Z -43.373,A 90.000,B 90.000,C 0.000} C_DIS
LIN {X 125.417,Y 21.431,Z -42.190,A 90.000,B 90.000,C 0.000} C_DIS
LIN {X 125.344,Y 21.431,Z -41.008,A 90.000,B 90.000,C 0.000} C_DIS
LIN {X 125.253,Y 21.431,Z -40.024,A 90.000,B 90.000,C 0.000} C_DIS
LIN {X 125.094,Y 21.431,Z -39.048,A 90.000,B 90.000,C 0.000} C_DIS
LIN {X 124.868,Y 21.431,Z -38.086,A 90.000,B 90.000,C 0.000} C_DIS
LIN {X 124.576,Y 21.431,Z -37.142,A 90.000,B 90.000,C 0.000} C_DIS
LIN {X 124.220,Y 21.431,Z -36.220,A 90.000,B 90.000,C 0.000} C_DIS
LIN {X 123.801,Y 21.431,Z -35.324,A 90.000,B 90.000,C 0.000} C_DIS
LIN {X 123.321,Y 21.431,Z -34.460,A 90.000,B 90.000,C 0.000} C_DIS
LIN {X 122.783,Y 21.431,Z -33.631,A 90.000,B 90.000,C 0.000} C_DIS
LIN {X 122.189,Y 21.431,Z -32.841,A 90.000,B 90.000,C 0.000} C_DIS
LIN {X 121.542,Y 21.431,Z -32.094,A 90.000,B 90.000,C 0.000} C_DIS
LIN {X 120.845,Y 21.431,Z -31.393,A 90.000,B 90.000,C 0.000} C_DIS
LIN {X 120.101,Y 21.431,Z -30.742,A 90.000,B 90.000,C 0.000} C_DIS
LIN {X 119.314,Y 21.431,Z -30.144,A 90.000,B 90.000,C 0.000} C_DIS
LIN {X 118.488,Y 21.431,Z -29.602,A 90.000,B 90.000,C 0.000} C_DIS
LIN {X 118.352,Y 21.431,Z -29.518,A 90.000,B 90.000,C 0.000} C_DIS
LIN {X 117.519,Y 21.431,Z -29.057,A 90.000,B 90.000,C 0.000} C_DIS
LIN {X 116.659,Y 21.431,Z -28.648,A 90.000,B 90.000,C 0.000} C_DIS
LIN {X 115.775,Y 21.431,Z -28.294,A 90.000,B 90.000,C 0.000} C_DIS
LIN {X 114.871,Y 21.431,Z -27.996,A 90.000,B 90.000,C 0.000} C_DIS
LIN {X 114.685,Y 21.431,Z -27.937,A 90.000,B 90.000,C 0.000} C_DIS
LIN {X 113.726,Y 21.431,Z -27.696,A 90.000,B 90.000,C 0.000} C_DIS
LIN {X 112.754,Y 21.431,Z -27.518,A 90.000,B 90.000,C 0.000} C_DIS
LIN {X 111.772,Y 21.431,Z -27.404,A 90.000,B 90.000,C 0.000} C_DIS
LIN {X 110.784,Y 21.431,Z -27.355,A 90.000,B 90.000,C 0.000} C_DIS
LIN {X 109.796,Y 21.431,Z -27.370,A 90.000,B 90.000,C 0.000} C_DIS
LIN {X 108.811,Y 21.431,Z -27.449,A 90.000,B 90.000,C 0.000} C_DIS
LIN {X 107.833,Y 21.431,Z -27.593,A 90.000,B 90.000,C 0.000} C_DIS
LIN {X 106.866,Y 21.431,Z -27.800,A 90.000,B 90.000,C 0.000} C_DIS
LIN {X 105.005,Y 21.431,Z -28.447,A 90.000,B 90.000,C 0.000} C_DIS
LIN {X 103.160,Y 21.431,Z -29.137,A 90.000,B 90.000,C 0.000} C_DIS
LIN {X 101.331,Y 21.431,Z -29.870,A 90.000,B 90.000,C 0.000} C_DIS
LIN {X 99.520,Y 21.431,Z -30.645,A 90.000,B 90.000,C 0.000} C_DIS
LIN {X 97.727,Y 21.431,Z -31.461,A 90.000,B 90.000,C 0.000} C_DIS
LIN {X 96.106,Y 21.431,Z -32.169,A 90.000,B 90.000,C 0.000} C_DIS
LIN {X 94.513,Y 21.431,Z -32.938,A 90.000,B 90.000,C 0.000} C_DIS
LIN {X 92.949,Y 21.431,Z -33.765,A 90.000,B 90.000,C 0.000} C_DIS
LIN {X 91.418,Y 21.431,Z -34.651,A 90.000,B 90.000,C 0.000} C_DIS
LIN {X 89.921,Y 21.431,Z -35.593,A 90.000,B 90.000,C 0.000} C_DIS
LIN {X 88.460,Y 21.431,Z -36.590,A 90.000,B 90.000,C 0.000} C_DIS
LIN {X 87.038,Y 21.431,Z -37.642,A 90.000,B 90.000,C 0.000} C_DIS
LIN {X 85.656,Y 21.431,Z -38.746,A 90.000,B 90.000,C 0.000} C_DIS
LIN {X 84.316,Y 21.431,Z -39.901,A 90.000,B 90.000,C 0.000} C_DIS
LIN {X 83.347,Y 21.431,Z -40.706,A 90.000,B 90.000,C 0.000} C_DIS
LIN {X 82.411,Y 21.431,Z -41.550,A 90.000,B 90.000,C 0.000} C_DIS
LIN {X 81.509,Y 21.431,Z -42.430,A 90.000,B 90.000,C 0.000} C_DIS
LIN {X 80.644,Y 21.431,Z -43.346,A 90.000,B 90.000,C 0.000} C_DIS
LIN {X 79.816,Y 21.431,Z -44.296,A 90.000,B 90.000,C 0.000} C_DIS
LIN {X 79.027,Y 21.431,Z -45.279,A 90.000,B 90.000,C 0.000} C_DIS
LIN {X 78.279,Y 21.431,Z -46.293,A 90.000,B 90.000,C 0.000} C_DIS
LIN {X 70.840,Y 21.431,Z -46.293,A 90.000,B 90.000,C 0.000} C_DIS
LIN {X 69.615,Y 21.431,Z -45.591,A 90.000,B 90.000,C 0.000} C_DIS
LIN {X 68.421,Y 21.431,Z -44.837,A 90.000,B 90.000,C 0.000} C_DIS
LIN {X 67.260,Y 21.431,Z -44.034,A 90.000,B 90.000,C 0.000} C_DIS
LIN {X 66.134,Y 21.431,Z -43.182,A 90.000,B 90.000,C 0.000} C_DIS
LIN {X 65.045,Y 21.431,Z -42.284,A 90.000,B 90.000,C 0.000} C_DIS
LIN {X 63.996,Y 21.431,Z -41.351,A 90.000,B 90.000,C 0.000} C_DIS
LIN {X 62.920,Y 21.431,Z -40.450,A 90.000,B 90.000,C 0.000} C_DIS
LIN {X 61.818,Y 21.431,Z -39.580,A 90.000,B 90.000,C 0.000} C_DIS
LIN {X 60.691,Y 21.431,Z -38.744,A 90.000,B 90.000,C 0.000} C_DIS
LIN {X 85.658,Y 21.431,Z -38.744,A 90.000,B 90.000,C 0.000} C_DIS
LIN {X 87.040,Y 21.431,Z -37.640,A 90.000,B 90.000,C 0.000} C_DIS
LIN {X 88.462,Y 21.431,Z -36.589,A 90.000,B 90.000,C 0.000} C_DIS
LIN {X 89.923,Y 21.431,Z -35.592,A 90.000,B 90.000,C 0.000} C_DIS
LIN {X 91.419,Y 21.431,Z -34.650,A 90.000,B 90.000,C 0.000} C_DIS
LIN {X 92.950,Y 21.431,Z -33.765,A 90.000,B 90.000,C 0.000} C_DIS
LIN {X 94.513,Y 21.431,Z -32.937,A 90.000,B 90.000,C 0.000} C_DIS
LIN {X 96.106,Y 21.431,Z -32.169,A 90.000,B 90.000,C 0.000} C_DIS
LIN {X 97.727,Y 21.431,Z -31.461,A 90.000,B 90.000,C 0.000} C_DIS
LIN {X 98.299,Y 21.431,Z -31.195,A 90.000,B 90.000,C 0.000} C_DIS
LIN {X 44.677,Y 21.431,Z -31.195,A 90.000,B 90.000,C 0.000} C_DIS
LIN {X 43.365,Y 21.431,Z -30.933,A 90.000,B 90.000,C 0.000} C_DIS
LIN {X 42.044,Y 21.431,Z -30.723,A 90.000,B 90.000,C 0.000} C_DIS
LIN {X 40.716,Y 21.431,Z -30.565,A 90.000,B 90.000,C 0.000} C_DIS
LIN {X 39.383,Y 21.431,Z -30.458,A 90.000,B 90.000,C 0.000} C_DIS
LIN {X 37.780,Y 21.431,Z -30.412,A 90.000,B 90.000,C 0.000} C_DIS
LIN {X 36.176,Y 21.431,Z -30.416,A 90.000,B 90.000,C 0.000} C_DIS
LIN {X 34.574,Y 21.431,Z -30.471,A 90.000,B 90.000,C 0.000} C_DIS
LIN {X 32.973,Y 21.431,Z -30.576,A 90.000,B 90.000,C 0.000} C_DIS
LIN {X 31.377,Y 21.431,Z -30.732,A 90.000,B 90.000,C 0.000} C_DIS
LIN {X 29.787,Y 21.431,Z -30.939,A 90.000,B 90.000,C 0.000} C_DIS
LIN {X 28.204,Y 21.431,Z -31.195,A 90.000,B 90.000,C 0.000} C_DIS
LIN {X -0.619,Y 21.431,Z -31.195,A 90.000,B 90.000,C 0.000} C_DIS
LIN {X 144.015,Y 21.431,Z -1.000,A 90.000,B 90.000,C 0.000} C_DIS
LIN {X -144.015,Y 21.431,Z -1.000,A 90.000,B 90.000,C 0.000} C_DIS
LIN {X -145.015,Y 21.431,Z 0.000,A 90.000,B 90.000,C 0.000} C_DIS
LIN {X 145.015,Y 21.431,Z 0.000,A 90.000,B 90.000,C 0.000} C_DIS
LIN {X 145.015,Y 21.431,Z -243.561,A 90.000,B 90.000,C 0.000} C_DIS
LIN {X 94.378,Y 21.431,Z -243.561,A 90.000,B 90.000,C 0.000} C_DIS
LIN {X 95.585,Y 21.431,Z -239.754,A 90.000,B 90.000,C 0.000} C_DIS
LIN {X 96.746,Y 21.431,Z -235.933,A 90.000,B 90.000,C 0.000} C_DIS
LIN {X 97.860,Y 21.431,Z -232.099,A 90.000,B 90.000,C 0.000} C_DIS
LIN {X 98.927,Y 21.431,Z -228.251,A 90.000,B 90.000,C 0.000} C_DIS
LIN {X 99.947,Y 21.431,Z -224.390,A 90.000,B 90.000,C 0.000} C_DIS
LIN {X 100.921,Y 21.431,Z -220.517,A 90.000,B 90.000,C 0.000} C_DIS
LIN {X 101.880,Y 21.431,Z -216.770,A 90.000,B 90.000,C 0.000} C_DIS
LIN {X 102.787,Y 21.431,Z -213.010,A 90.000,B 90.000,C 0.000} C_DIS
LIN {X 103.643,Y 21.431,Z -209.237,A 90.000,B 90.000,C 0.000} C_DIS
LIN {X 104.447,Y 21.431,Z -205.454,A 90.000,B 90.000,C 0.000} C_DIS
LIN {X 105.198,Y 21.431,Z -201.660,A 90.000,B 90.000,C 0.000} C_DIS
LIN {X 105.898,Y 21.431,Z -197.855,A 90.000,B 90.000,C 0.000} C_DIS
LIN {X 106.546,Y 21.431,Z -194.042,A 90.000,B 90.000,C 0.000} C_DIS
LIN {X 107.141,Y 21.431,Z -190.220,A 90.000,B 90.000,C 0.000} C_DIS
LIN {X 107.970,Y 21.431,Z -184.477,A 90.000,B 90.000,C 0.000} C_DIS
LIN {X 108.736,Y 21.431,Z -178.724,A 90.000,B 90.000,C 0.000} C_DIS
LIN {X 109.438,Y 21.431,Z -172.964,A 90.000,B 90.000,C 0.000} C_DIS
LIN {X 110.077,Y 21.431,Z -167.196,A 90.000,B 90.000,C 0.000} C_DIS
LIN {X 110.652,Y 21.431,Z -161.422,A 90.000,B 90.000,C 0.000} C_DIS
LIN {X 111.163,Y 21.431,Z -155.642,A 90.000,B 90.000,C 0.000} C_DIS
LIN {X 111.610,Y 21.431,Z -149.856,A 90.000,B 90.000,C 0.000} C_DIS
LIN {X 111.854,Y 21.431,Z -146.867,A 90.000,B 90.000,C 0.000} C_DIS
LIN {X 112.045,Y 21.431,Z -143.875,A 90.000,B 90.000,C 0.000} C_DIS
LIN {X 112.182,Y 21.431,Z -140.879,A 90.000,B 90.000,C 0.000} C_DIS
LIN {X 112.266,Y 21.431,Z -137.882,A 90.000,B 90.000,C 0.000} C_DIS
LIN {X 112.296,Y 21.431,Z -134.883,A 90.000,B 90.000,C 0.000} C_DIS
LIN {X 112.273,Y 21.431,Z -131.885,A 90.000,B 90.000,C 0.000} C_DIS
LIN {X 112.196,Y 21.431,Z -128.887,A 90.000,B 90.000,C 0.000} C_DIS
LIN {X 112.066,Y 21.431,Z -125.891,A 90.000,B 90.000,C 0.000} C_DIS
LIN {X 111.675,Y 21.431,Z -121.469,A 90.000,B 90.000,C 0.000} C_DIS
LIN {X 111.228,Y 21.431,Z -117.051,A 90.000,B 90.000,C 0.000} C_DIS
LIN {X 110.726,Y 21.431,Z -112.640,A 90.000,B 90.000,C 0.000} C_DIS
LIN {X 110.168,Y 21.431,Z -108.236,A 90.000,B 90.000,C 0.000} C_DIS
LIN {X 109.556,Y 21.431,Z -103.838,A 90.000,B 90.000,C 0.000} C_DIS
LIN {X 108.888,Y 21.431,Z -99.449,A 90.000,B 90.000,C 0.000} C_DIS
LIN {X 108.872,Y 21.431,Z -99.264,A 90.000,B 90.000,C 0.000} C_DIS
LIN {X 108.683,Y 21.431,Z -98.020,A 90.000,B 90.000,C 0.000} C_DIS
LIN {X 108.676,Y 21.431,Z -97.926,A 90.000,B 90.000,C 0.000} C_DIS
LIN {X 108.433,Y 21.431,Z -96.043,A 90.000,B 90.000,C 0.000} C_DIS
LIN {X 108.133,Y 21.431,Z -94.169,A 90.000,B 90.000,C 0.000} C_DIS
LIN {X 107.777,Y 21.431,Z -92.304,A 90.000,B 90.000,C 0.000} C_DIS
LIN {X 107.364,Y 21.431,Z -90.451,A 90.000,B 90.000,C 0.000} C_DIS
LIN {X 107.109,Y 21.431,Z -89.911,A 90.000,B 90.000,C 0.000} C_DIS
LIN {X 106.908,Y 21.431,Z -89.348,A 90.000,B 90.000,C 0.000} C_DIS
LIN {X 106.764,Y 21.431,Z -88.769,A 90.000,B 90.000,C 0.000} C_DIS
LIN {X 106.678,Y 21.431,Z -88.178,A 90.000,B 90.000,C 0.000} C_DIS
LIN {X 106.649,Y 21.431,Z -87.581,A 90.000,B 90.000,C 0.000} C_DIS
LIN {X 107.930,Y 21.431,Z -85.625,A 90.000,B 90.000,C 0.000} C_DIS
LIN {X 109.151,Y 21.431,Z -83.631,A 90.000,B 90.000,C 0.000} C_DIS
LIN {X 110.309,Y 21.431,Z -81.600,A 90.000,B 90.000,C 0.000} C_DIS
LIN {X 111.404,Y 21.431,Z -79.535,A 90.000,B 90.000,C 0.000} C_DIS
LIN {X 112.435,Y 21.431,Z -77.436,A 90.000,B 90.000,C 0.000} C_DIS
LIN {X 113.401,Y 21.431,Z -75.307,A 90.000,B 90.000,C 0.000} C_DIS
LIN {X 114.300,Y 21.431,Z -73.149,A 90.000,B 90.000,C 0.000} C_DIS
LIN {X 115.133,Y 21.431,Z -70.964,A 90.000,B 90.000,C 0.000} C_DIS
LIN {X 115.897,Y 21.431,Z -68.755,A 90.000,B 90.000,C 0.000} C_DIS
LIN {X 116.594,Y 21.431,Z -66.523,A 90.000,B 90.000,C 0.000} C_DIS
LIN {X 117.391,Y 21.431,Z -63.629,A 90.000,B 90.000,C 0.000} C_DIS
LIN {X 118.216,Y 21.431,Z -60.743,A 90.000,B 90.000,C 0.000} C_DIS
LIN {X 118.900,Y 21.431,Z -58.947,A 90.000,B 90.000,C 0.000} C_DIS
LIN {X 119.632,Y 21.431,Z -57.170,A 90.000,B 90.000,C 0.000} C_DIS
LIN {X 120.411,Y 21.431,Z -55.413,A 90.000,B 90.000,C 0.000} C_DIS
LIN {X 121.238,Y 21.431,Z -53.679,A 90.000,B 90.000,C 0.000} C_DIS
LIN {X 122.112,Y 21.431,Z -51.967,A 90.000,B 90.000,C 0.000} C_DIS
LIN {X 122.620,Y 21.431,Z -50.961,A 90.000,B 90.000,C 0.000} C_DIS
LIN {X 123.069,Y 21.431,Z -49.926,A 90.000,B 90.000,C 0.000} C_DIS
LIN {X 123.455,Y 21.431,Z -48.867,A 90.000,B 90.000,C 0.000} C_DIS
LIN {X 123.778,Y 21.431,Z -47.788,A 90.000,B 90.000,C 0.000} C_DIS
LIN {X 124.038,Y 21.431,Z -46.690,A 90.000,B 90.000,C 0.000} C_DIS
LIN {X 124.232,Y 21.431,Z -45.580,A 90.000,B 90.000,C 0.000} C_DIS
LIN {X 124.360,Y 21.431,Z -44.460,A 90.000,B 90.000,C 0.000} C_DIS
LIN {X 124.422,Y 21.431,Z -43.334,A 90.000,B 90.000,C 0.000} C_DIS
LIN {X 124.417,Y 21.431,Z -42.207,A 90.000,B 90.000,C 0.000} C_DIS
LIN {X 124.347,Y 21.431,Z -41.082,A 90.000,B 90.000,C 0.000} C_DIS
LIN {X 124.254,Y 21.431,Z -40.095,A 90.000,B 90.000,C 0.000} C_DIS
LIN {X 124.088,Y 21.431,Z -39.117,A 90.000,B 90.000,C 0.000} C_DIS
LIN {X 123.849,Y 21.431,Z -38.155,A 90.000,B 90.000,C 0.000} C_DIS
LIN {X 123.540,Y 21.431,Z -37.213,A 90.000,B 90.000,C 0.000} C_DIS
LIN {X 123.161,Y 21.431,Z -36.296,A 90.000,B 90.000,C 0.000} C_DIS
LIN {X 122.715,Y 21.431,Z -35.411,A 90.000,B 90.000,C 0.000} C_DIS
LIN {X 122.205,Y 21.431,Z -34.561,A 90.000,B 90.000,C 0.000} C_DIS
LIN {X 121.633,Y 21.431,Z -33.751,A 90.000,B 90.000,C 0.000} C_DIS
LIN {X 121.002,Y 21.431,Z -32.986,A 90.000,B 90.000,C 0.000} C_DIS
LIN {X 120.316,Y 21.431,Z -32.270,A 90.000,B 90.000,C 0.000} C_DIS
LIN {X 119.578,Y 21.431,Z -31.607,A 90.000,B 90.000,C 0.000} C_DIS
LIN {X 118.794,Y 21.431,Z -31.001,A 90.000,B 90.000,C 0.000} C_DIS
LIN {X 117.966,Y 21.431,Z -30.455,A 90.000,B 90.000,C 0.000} C_DIS
LIN {X 117.834,Y 21.431,Z -30.373,A 90.000,B 90.000,C 0.000} C_DIS
LIN {X 117.055,Y 21.431,Z -29.942,A 90.000,B 90.000,C 0.000} C_DIS
LIN {X 116.250,Y 21.431,Z -29.561,A 90.000,B 90.000,C 0.000} C_DIS
LIN {X 115.424,Y 21.431,Z -29.230,A 90.000,B 90.000,C 0.000} C_DIS
LIN {X 114.578,Y 21.431,Z -28.952,A 90.000,B 90.000,C 0.000} C_DIS
LIN {X 114.396,Y 21.431,Z -28.894,A 90.000,B 90.000,C 0.000} C_DIS
LIN {X 113.507,Y 21.431,Z -28.671,A 90.000,B 90.000,C 0.000} C_DIS
LIN {X 112.605,Y 21.431,Z -28.507,A 90.000,B 90.000,C 0.000} C_DIS
LIN {X 111.695,Y 21.431,Z -28.401,A 90.000,B 90.000,C 0.000} C_DIS
LIN {X 110.779,Y 21.431,Z -28.354,A 90.000,B 90.000,C 0.000} C_DIS
LIN {X 109.863,Y 21.431,Z -28.367,A 90.000,B 90.000,C 0.000} C_DIS
LIN {X 108.949,Y 21.431,Z -28.439,A 90.000,B 90.000,C 0.000} C_DIS
LIN {X 108.042,Y 21.431,Z -28.571,A 90.000,B 90.000,C 0.000} C_DIS
LIN {X 107.145,Y 21.431,Z -28.761,A 90.000,B 90.000,C 0.000} C_DIS
LIN {X 105.310,Y 21.431,Z -29.400,A 90.000,B 90.000,C 0.000} C_DIS
LIN {X 103.490,Y 21.431,Z -30.082,A 90.000,B 90.000,C 0.000} C_DIS
LIN {X 101.686,Y 21.431,Z -30.805,A 90.000,B 90.000,C 0.000} C_DIS
LIN {X 99.899,Y 21.431,Z -31.570,A 90.000,B 90.000,C 0.000} C_DIS
LIN {X 98.131,Y 21.431,Z -32.376,A 90.000,B 90.000,C 0.000} C_DIS
LIN {X 96.539,Y 21.431,Z -33.071,A 90.000,B 90.000,C 0.000} C_DIS
LIN {X 94.974,Y 21.431,Z -33.825,A 90.000,B 90.000,C 0.000} C_DIS
LIN {X 93.439,Y 21.431,Z -34.637,A 90.000,B 90.000,C 0.000} C_DIS
LIN {X 91.935,Y 21.431,Z -35.507,A 90.000,B 90.000,C 0.000} C_DIS
LIN {X 90.465,Y 21.431,Z -36.432,A 90.000,B 90.000,C 0.000} C_DIS
LIN {X 89.030,Y 21.431,Z -37.412,A 90.000,B 90.000,C 0.000} C_DIS
LIN {X 87.634,Y 21.431,Z -38.445,A 90.000,B 90.000,C 0.000} C_DIS
LIN {X 86.277,Y 21.431,Z -39.530,A 90.000,B 90.000,C 0.000} C_DIS
LIN {X 84.962,Y 21.431,Z -40.665,A 90.000,B 90.000,C 0.000} C_DIS
LIN {X 83.832,Y 21.431,Z -41.610,A 90.000,B 90.000,C 0.000} C_DIS
LIN {X 82.749,Y 21.431,Z -42.608,A 90.000,B 90.000,C 0.000} C_DIS
LIN {X 81.716,Y 21.431,Z -43.658,A 90.000,B 90.000,C 0.000} C_DIS
LIN {X 80.736,Y 21.431,Z -44.757,A 90.000,B 90.000,C 0.000} C_DIS
LIN {X 79.810,Y 21.431,Z -45.903,A 90.000,B 90.000,C 0.000} C_DIS
LIN {X 78.940,Y 21.431,Z -47.092,A 90.000,B 90.000,C 0.000} C_DIS
LIN {X 78.130,Y 21.431,Z -48.321,A 90.000,B 90.000,C 0.000} C_DIS
LIN {X 77.380,Y 21.431,Z -49.589,A 90.000,B 90.000,C 0.000} C_DIS
LIN {X 76.693,Y 21.431,Z -50.892,A 90.000,B 90.000,C 0.000} C_DIS
LIN {X 75.312,Y 21.431,Z -50.014,A 90.000,B 90.000,C 0.000} C_DIS
LIN {X 73.914,Y 21.431,Z -49.163,A 90.000,B 90.000,C 0.000} C_DIS
LIN {X 72.500,Y 21.431,Z -48.340,A 90.000,B 90.000,C 0.000} C_DIS
LIN {X 71.069,Y 21.431,Z -47.546,A 90.000,B 90.000,C 0.000} C_DIS
LIN {X 69.884,Y 21.431,Z -46.905,A 90.000,B 90.000,C 0.000} C_DIS
LIN {X 68.724,Y 21.431,Z -46.217,A 90.000,B 90.000,C 0.000} C_DIS
LIN {X 67.593,Y 21.431,Z -45.485,A 90.000,B 90.000,C 0.000} C_DIS
LIN {X 66.490,Y 21.431,Z -44.709,A 90.000,B 90.000,C 0.000} C_DIS
LIN {X 65.420,Y 21.431,Z -43.891,A 90.000,B 90.000,C 0.000} C_DIS
LIN {X 64.381,Y 21.431,Z -43.032,A 90.000,B 90.000,C 0.000} C_DIS
LIN {X 63.151,Y 21.431,Z -41.943,A 90.000,B 90.000,C 0.000} C_DIS
LIN {X 61.882,Y 21.431,Z -40.898,A 90.000,B 90.000,C 0.000} C_DIS
LIN {X 60.578,Y 21.431,Z -39.899,A 90.000,B 90.000,C 0.000} C_DIS
LIN {X 59.239,Y 21.431,Z -38.947,A 90.000,B 90.000,C 0.000} C_DIS
LIN {X 57.867,Y 21.431,Z -38.044,A 90.000,B 90.000,C 0.000} C_DIS
LIN {X 56.463,Y 21.431,Z -37.189,A 90.000,B 90.000,C 0.000} C_DIS
LIN {X 55.030,Y 21.431,Z -36.385,A 90.000,B 90.000,C 0.000} C_DIS
LIN {X 53.570,Y 21.431,Z -35.632,A 90.000,B 90.000,C 0.000} C_DIS
LIN {X 52.248,Y 21.431,Z -34.931,A 90.000,B 90.000,C 0.000} C_DIS
LIN {X 50.896,Y 21.431,Z -34.291,A 90.000,B 90.000,C 0.000} C_DIS
LIN {X 49.516,Y 21.431,Z -33.712,A 90.000,B 90.000,C 0.000} C_DIS
LIN {X 48.111,Y 21.431,Z -33.195,A 90.000,B 90.000,C 0.000} C_DIS
LIN {X 46.685,Y 21.431,Z -32.742,A 90.000,B 90.000,C 0.000} C_DIS
LIN {X 45.240,Y 21.431,Z -32.353,A 90.000,B 90.000,C 0.000} C_DIS
LIN {X 43.779,Y 21.431,Z -32.030,A 90.000,B 90.000,C 0.000} C_DIS
LIN {X 42.305,Y 21.431,Z -31.772,A 90.000,B 90.000,C 0.000} C_DIS
LIN {X 40.821,Y 21.431,Z -31.581,A 90.000,B 90.000,C 0.000} C_DIS
LIN {X 39.330,Y 21.431,Z -31.457,A 90.000,B 90.000,C 0.000} C_DIS
LIN {X 37.492,Y 21.431,Z -31.409,A 90.000,B 90.000,C 0.000} C_DIS
LIN {X 35.654,Y 21.431,Z -31.429,A 90.000,B 90.000,C 0.000} C_DIS
LIN {X 33.817,Y 21.431,Z -31.517,A 90.000,B 90.000,C 0.000} C_DIS
LIN {X 31.985,Y 21.431,Z -31.673,A 90.000,B 90.000,C 0.000} C_DIS
LIN {X 30.160,Y 21.431,Z -31.896,A 90.000,B 90.000,C 0.000} C_DIS
LIN {X 28.345,Y 21.431,Z -32.186,A 90.000,B 90.000,C 0.000} C_DIS
LIN {X 26.541,Y 21.431,Z -32.543,A 90.000,B 90.000,C 0.000} C_DIS
LIN {X 25.192,Y 21.431,Z -32.853,A 90.000,B 90.000,C 0.000} C_DIS
LIN {X 23.830,Y 21.431,Z -33.100,A 90.000,B 90.000,C 0.000} C_DIS
LIN {X 22.459,Y 21.431,Z -33.284,A 90.000,B 90.000,C 0.000} C_DIS
LIN {X 21.080,Y 21.431,Z -33.405,A 90.000,B 90.000,C 0.000} C_DIS
LIN {X 19.697,Y 21.431,Z -33.461,A 90.000,B 90.000,C 0.000} C_DIS
LIN {X 18.313,Y 21.431,Z -33.454,A 90.000,B 90.000,C 0.000} C_DIS
LIN {X 14.507,Y 21.431,Z -33.082,A 90.000,B 90.000,C 0.000} C_DIS
LIN {X 10.697,Y 21.431,Z -32.738,A 90.000,B 90.000,C 0.000} C_DIS
LIN {X 6.886,Y 21.431,Z -32.421,A 90.000,B 90.000,C 0.000} C_DIS
LIN {X 5.110,Y 21.431,Z -32.454,A 90.000,B 90.000,C 0.000} C_DIS
LIN {X 3.335,Y 21.431,Z -32.434,A 90.000,B 90.000,C 0.000} C_DIS
LIN {X 1.560,Y 21.431,Z -32.361,A 90.000,B 90.000,C 0.000} C_DIS
LIN {X -0.211,Y 21.431,Z -32.236,A 90.000,B 90.000,C 0.000} C_DIS
LIN {X -1.978,Y 21.431,Z -32.058,A 90.000,B 90.000,C 0.000} C_DIS
LIN {X -3.870,Y 21.431,Z -31.612,A 90.000,B 90.000,C 0.000} C_DIS
LIN {X -5.753,Y 21.431,Z -31.127,A 90.000,B 90.000,C 0.000} C_DIS
LIN {X -7.626,Y 21.431,Z -30.604,A 90.000,B 90.000,C 0.000} C_DIS
LIN {X -9.487,Y 21.431,Z -30.041,A 90.000,B 90.000,C 0.000} C_DIS
LIN {X -12.387,Y 21.431,Z -29.299,A 90.000,B 90.000,C 0.000} C_DIS
LIN {X -15.300,Y 21.431,Z -28.609,A 90.000,B 90.000,C 0.000} C_DIS
LIN {X -18.226,Y 21.431,Z -27.972,A 90.000,B 90.000,C 0.000} C_DIS
LIN {X -21.162,Y 21.431,Z -27.387,A 90.000,B 90.000,C 0.000} C_DIS
LIN {X -24.107,Y 21.431,Z -26.854,A 90.000,B 90.000,C 0.000} C_DIS
LIN {X -27.063,Y 21.431,Z -26.374,A 90.000,B 90.000,C 0.000} C_DIS
LIN {X -30.026,Y 21.431,Z -25.948,A 90.000,B 90.000,C 0.000} C_DIS
LIN {X -32.996,Y 21.431,Z -25.574,A 90.000,B 90.000,C 0.000} C_DIS
LIN {X -36.315,Y 21.431,Z -25.329,A 90.000,B 90.000,C 0.000} C_DIS
LIN {X -39.638,Y 21.431,Z -25.134,A 90.000,B 90.000,C 0.000} C_DIS
LIN {X -42.963,Y 21.431,Z -24.989,A 90.000,B 90.000,C 0.000} C_DIS
LIN {X -46.290,Y 21.431,Z -24.895,A 90.000,B 90.000,C 0.000} C_DIS
LIN {X -47.917,Y 21.431,Z -24.787,A 90.000,B 90.000,C 0.000} C_DIS
LIN {X -49.545,Y 21.431,Z -24.710,A 90.000,B 90.000,C 0.000} C_DIS
LIN {X -49.699,Y 21.431,Z -24.725,A 90.000,B 90.000,C 0.000} C_DIS
LIN {X -51.070,Y 21.431,Z -24.620,A 90.000,B 90.000,C 0.000} C_DIS
LIN {X -52.434,Y 21.431,Z -24.457,A 90.000,B 90.000,C 0.000} C_DIS
LIN {X -53.791,Y 21.431,Z -24.236,A 90.000,B 90.000,C 0.000} C_DIS
LIN {X -55.137,Y 21.431,Z -23.957,A 90.000,B 90.000,C 0.000} C_DIS
LIN {X -56.470,Y 21.431,Z -23.621,A 90.000,B 90.000,C 0.000} C_DIS
LIN {X -57.787,Y 21.431,Z -23.228,A 90.000,B 90.000,C 0.000} C_DIS
LIN {X -57.835,Y 21.431,Z -23.114,A 90.000,B 90.000,C 0.000} C_DIS
LIN {X -58.293,Y 21.431,Z -22.144,A 90.000,B 90.000,C 0.000} C_DIS
LIN {X -58.781,Y 21.431,Z -21.189,A 90.000,B 90.000,C 0.000} C_DIS
LIN {X -59.298,Y 21.431,Z -20.250,A 90.000,B 90.000,C 0.000} C_DIS
LIN {X -60.095,Y 21.431,Z -19.160,A 90.000,B 90.000,C 0.000} C_DIS
LIN {X -60.946,Y 21.431,Z -18.111,A 90.000,B 90.000,C 0.000} C_DIS
LIN {X -61.849,Y 21.431,Z -17.107,A 90.000,B 90.000,C 0.000} C_DIS
LIN {X -62.802,Y 21.431,Z -16.149,A 90.000,B 90.000,C 0.000} C_DIS
LIN {X -63.801,Y 21.431,Z -15.240,A 90.000,B 90.000,C 0.000} C_DIS
LIN {X -64.845,Y 21.431,Z -14.384,A 90.000,B 90.000,C 0.000} C_DIS
LIN {X -65.931,Y 21.431,Z -13.580,A 90.000,B 90.000,C 0.000} C_DIS
LIN {X -67.056,Y 21.431,Z -12.833,A 90.000,B 90.000,C 0.000} C_DIS
LIN {X -68.218,Y 21.431,Z -12.143,A 90.000,B 90.000,C 0.000} C_DIS
LIN {X -69.412,Y 21.431,Z -11.513,A 90.000,B 90.000,C 0.000} C_DIS
LIN {X -70.637,Y 21.431,Z -10.944,A 90.000,B 90.000,C 0.000} C_DIS
LIN {X -71.889,Y 21.431,Z -10.437,A 90.000,B 90.000,C 0.000} C_DIS
LIN {X -73.165,Y 21.431,Z -9.994,A 90.000,B 90.000,C 0.000} C_DIS
LIN {X -74.159,Y 21.431,Z -9.691,A 90.000,B 90.000,C 0.000} C_DIS
LIN {X -75.171,Y 21.431,Z -9.455,A 90.000,B 90.000,C 0.000} C_DIS
LIN {X -76.196,Y 21.431,Z -9.288,A 90.000,B 90.000,C 0.000} C_DIS
LIN {X -77.231,Y 21.431,Z -9.191,A 90.000,B 90.000,C 0.000} C_DIS
LIN {X -78.269,Y 21.431,Z -9.164,A 90.000,B 90.000,C 0.000} C_DIS
LIN {X -79.307,Y 21.431,Z -9.207,A 90.000,B 90.000,C 0.000} C_DIS
LIN {X -80.340,Y 21.431,Z -9.320,A 90.000,B 90.000,C 0.000} C_DIS
LIN {X -81.363,Y 21.431,Z -9.502,A 90.000,B 90.000,C 0.000} C_DIS
LIN {X -82.371,Y 21.431,Z -9.753,A 90.000,B 90.000,C 0.000} C_DIS
LIN {X -83.361,Y 21.431,Z -10.071,A 90.000,B 90.000,C 0.000} C_DIS
LIN {X -84.326,Y 21.431,Z -10.455,A 90.000,B 90.000,C 0.000} C_DIS
LIN {X -85.263,Y 21.431,Z -10.904,A 90.000,B 90.000,C 0.000} C_DIS
LIN {X -86.036,Y 21.431,Z -11.312,A 90.000,B 90.000,C 0.000} C_DIS
LIN {X -86.777,Y 21.431,Z -11.775,A 90.000,B 90.000,C 0.000} C_DIS
LIN {X -87.483,Y 21.431,Z -12.290,A 90.000,B 90.000,C 0.000} C_DIS
LIN {X -88.150,Y 21.431,Z -12.855,A 90.000,B 90.000,C 0.000} C_DIS
LIN {X -88.775,Y 21.431,Z -13.467,A 90.000,B 90.000,C 0.000} C_DIS
LIN {X -89.354,Y 21.431,Z -14.122,A 90.000,B 90.000,C 0.000} C_DIS
LIN {X -89.884,Y 21.431,Z -14.817,A 90.000,B 90.000,C 0.000} C_DIS
LIN {X -90.362,Y 21.431,Z -15.549,A 90.000,B 90.000,C 0.000} C_DIS
LIN {X -90.786,Y 21.431,Z -16.313,A 90.000,B 90.000,C 0.000} C_DIS
LIN {X -91.154,Y 21.431,Z -17.106,A 90.000,B 90.000,C 0.000} C_DIS
LIN {X -91.464,Y 21.431,Z -17.923,A 90.000,B 90.000,C 0.000} C_DIS
LIN {X -92.399,Y 21.431,Z -17.891,A 90.000,B 90.000,C 0.000} C_DIS
LIN {X -93.335,Y 21.431,Z -17.920,A 90.000,B 90.000,C 0.000} C_DIS
LIN {X -94.266,Y 21.431,Z -18.009,A 90.000,B 90.000,C 0.000} C_DIS
LIN {X -95.190,Y 21.431,Z -18.158,A 90.000,B 90.000,C 0.000} C_DIS
LIN {X -96.102,Y 21.431,Z -18.367,A 90.000,B 90.000,C 0.000} C_DIS
LIN {X -96.999,Y 21.431,Z -18.634,A 90.000,B 90.000,C 0.000} C_DIS
LIN {X -97.145,Y 21.431,Z -18.687,A 90.000,B 90.000,C 0.000} C_DIS
LIN {X -97.843,Y 21.431,Z -18.957,A 90.000,B 90.000,C 0.000} C_DIS
LIN {X -98.520,Y 21.431,Z -19.275,A 90.000,B 90.000,C 0.000} C_DIS
LIN {X -99.174,Y 21.431,Z -19.639,A 90.000,B 90.000,C 0.000} C_DIS
LIN {X -99.801,Y 21.431,Z -20.047,A 90.000,B 90.000,C 0.000} C_DIS
LIN {X -99.964,Y 21.431,Z -20.159,A 90.000,B 90.000,C 0.000} C_DIS
LIN {X -100.786,Y 21.431,Z -20.800,A 90.000,B 90.000,C 0.000} C_DIS
LIN {X -101.566,Y 21.431,Z -21.491,A 90.000,B 90.000,C 0.000} C_DIS
LIN {X -102.303,Y 21.431,Z -22.228,A 90.000,B 90.000,C 0.000} C_DIS
LIN {X -102.993,Y 21.431,Z -23.010,A 90.000,B 90.000,C 0.000} C_DIS
LIN {X -103.633,Y 21.431,Z -23.832,A 90.000,B 90.000,C 0.000} C_DIS
LIN {X -104.222,Y 21.431,Z -24.692,A 90.000,B 90.000,C 0.000} C_DIS
LIN {X -104.756,Y 21.431,Z -25.587,A 90.000,B 90.000,C 0.000} C_DIS
LIN {X -104.823,Y 21.431,Z -25.846,A 90.000,B 90.000,C 0.000} C_DIS
LIN {X -104.937,Y 21.431,Z -26.088,A 90.000,B 90.000,C 0.000} C_DIS
LIN {X -105.096,Y 21.431,Z -26.304,A 90.000,B 90.000,C 0.000} C_DIS
LIN {X -105.292,Y 21.431,Z -26.485,A 90.000,B 90.000,C 0.000} C_DIS
LIN {X -105.519,Y 21.431,Z -26.627,A 90.000,B 90.000,C 0.000} C_DIS
LIN {X -105.769,Y 21.431,Z -26.722,A 90.000,B 90.000,C 0.000} C_DIS
LIN {X -106.610,Y 21.431,Z -27.155,A 90.000,B 90.000,C 0.000} C_DIS
LIN {X -107.421,Y 21.431,Z -27.642,A 90.000,B 90.000,C 0.000} C_DIS
LIN {X -108.197,Y 21.431,Z -28.182,A 90.000,B 90.000,C 0.000} C_DIS
LIN {X -108.936,Y 21.431,Z -28.772,A 90.000,B 90.000,C 0.000} C_DIS
LIN {X -109.634,Y 21.431,Z -29.410,A 90.000,B 90.000,C 0.000} C_DIS
LIN {X -110.288,Y 21.431,Z -30.093,A 90.000,B 90.000,C 0.000} C_DIS
LIN {X -110.958,Y 21.431,Z -30.408,A 90.000,B 90.000,C 0.000} C_DIS
LIN {X -111.605,Y 21.431,Z -30.769,A 90.000,B 90.000,C 0.000} C_DIS
LIN {X -112.225,Y 21.431,Z -31.174,A 90.000,B 90.000,C 0.000} C_DIS
LIN {X -112.315,Y 21.431,Z -31.236,A 90.000,B 90.000,C 0.000} C_DIS
LIN {X -113.450,Y 21.431,Z -32.156,A 90.000,B 90.000,C 0.000} C_DIS
LIN {X -113.584,Y 21.431,Z -32.281,A 90.000,B 90.000,C 0.000} C_DIS
LIN {X -114.151,Y 21.431,Z -32.848,A 90.000,B 90.000,C 0.000} C_DIS
LIN {X -114.678,Y 21.431,Z -33.452,A 90.000,B 90.000,C 0.000} C_DIS
LIN {X -115.163,Y 21.431,Z -34.090,A 90.000,B 90.000,C 0.000} C_DIS
LIN {X -115.604,Y 21.431,Z -34.760,A 90.000,B 90.000,C 0.000} C_DIS
LIN {X -115.680,Y 21.431,Z -34.882,A 90.000,B 90.000,C 0.000} C_DIS
LIN {X -116.417,Y 21.431,Z -36.303,A 90.000,B 90.000,C 0.000} C_DIS
LIN {X -116.760,Y 21.431,Z -37.258,A 90.000,B 90.000,C 0.000} C_DIS
LIN {X -117.041,Y 21.431,Z -38.233,A 90.000,B 90.000,C 0.000} C_DIS
LIN {X -117.261,Y 21.431,Z -39.223,A 90.000,B 90.000,C 0.000} C_DIS
LIN {X -117.417,Y 21.431,Z -40.226,A 90.000,B 90.000,C 0.000} C_DIS
LIN {X -117.509,Y 21.431,Z -41.236,A 90.000,B 90.000,C 0.000} C_DIS
LIN {X -117.537,Y 21.431,Z -42.250,A 90.000,B 90.000,C 0.000} C_DIS
LIN {X -117.501,Y 21.431,Z -43.264,A 90.000,B 90.000,C 0.000} C_DIS
LIN {X -117.401,Y 21.431,Z -44.274,A 90.000,B 90.000,C 0.000} C_DIS
LIN {X -117.236,Y 21.431,Z -45.275,A 90.000,B 90.000,C 0.000} C_DIS
LIN {X -117.009,Y 21.431,Z -46.264,A 90.000,B 90.000,C 0.000} C_DIS
LIN {X -116.720,Y 21.431,Z -47.236,A 90.000,B 90.000,C 0.000} C_DIS
LIN {X -116.369,Y 21.431,Z -48.188,A 90.000,B 90.000,C 0.000} C_DIS
LIN {X -116.484,Y 21.431,Z -48.721,A 90.000,B 90.000,C 0.000} C_DIS
LIN {X -116.556,Y 21.431,Z -49.261,A 90.000,B 90.000,C 0.000} C_DIS
LIN {X -116.588,Y 21.431,Z -50.386,A 90.000,B 90.000,C 0.000} C_DIS
LIN {X -116.548,Y 21.431,Z -51.510,A 90.000,B 90.000,C 0.000} C_DIS
LIN {X -116.438,Y 21.431,Z -52.630,A 90.000,B 90.000,C 0.000} C_DIS
LIN {X -116.258,Y 21.431,Z -53.741,A 90.000,B 90.000,C 0.000} C_DIS
LIN {X -116.007,Y 21.431,Z -54.838,A 90.000,B 90.000,C 0.000} C_DIS
LIN {X -115.689,Y 21.431,Z -55.917,A 90.000,B 90.000,C 0.000} C_DIS
LIN {X -115.303,Y 21.431,Z -56.974,A 90.000,B 90.000,C 0.000} C_DIS
LIN {X -114.851,Y 21.431,Z -58.005,A 90.000,B 90.000,C 0.000} C_DIS
LIN {X -114.335,Y 21.431,Z -59.005,A 90.000,B 90.000,C 0.000} C_DIS
LIN {X -113.757,Y 21.431,Z -59.970,A 90.000,B 90.000,C 0.000} C_DIS
LIN {X -113.119,Y 21.431,Z -60.897,A 90.000,B 90.000,C 0.000} C_DIS
LIN {X -111.807,Y 21.431,Z -62.498,A 90.000,B 90.000,C 0.000} C_DIS
LIN {X -110.443,Y 21.431,Z -64.055,A 90.000,B 90.000,C 0.000} C_DIS
LIN {X -109.028,Y 21.431,Z -65.567,A 90.000,B 90.000,C 0.000} C_DIS
LIN {X -107.565,Y 21.431,Z -67.031,A 90.000,B 90.000,C 0.000} C_DIS
LIN {X -106.055,Y 21.431,Z -68.447,A 90.000,B 90.000,C 0.000} C_DIS
LIN {X -104.499,Y 21.431,Z -69.813,A 90.000,B 90.000,C 0.000} C_DIS
LIN {X -102.900,Y 21.431,Z -71.126,A 90.000,B 90.000,C 0.000} C_DIS
LIN {X -101.258,Y 21.431,Z -72.387,A 90.000,B 90.000,C 0.000} C_DIS
LIN {X -99.576,Y 21.431,Z -73.594,A 90.000,B 90.000,C 0.000} C_DIS
LIN {X -97.461,Y 21.431,Z -74.900,A 90.000,B 90.000,C 0.000} C_DIS
LIN {X -95.359,Y 21.431,Z -76.228,A 90.000,B 90.000,C 0.000} C_DIS
LIN {X -95.223,Y 21.431,Z -76.304,A 90.000,B 90.000,C 0.000} C_DIS
LIN {X -94.952,Y 21.431,Z -76.493,A 90.000,B 90.000,C 0.000} C_DIS
LIN {X -94.692,Y 21.431,Z -76.699,A 90.000,B 90.000,C 0.000} C_DIS
LIN {X -94.446,Y 21.431,Z -76.920,A 90.000,B 90.000,C 0.000} C_DIS
LIN {X -94.344,Y 21.431,Z -76.997,A 90.000,B 90.000,C 0.000} C_DIS
LIN {X -93.709,Y 21.431,Z -77.538,A 90.000,B 90.000,C 0.000} C_DIS
LIN {X -93.064,Y 21.431,Z -78.068,A 90.000,B 90.000,C 0.000} C_DIS
LIN {X -91.856,Y 21.431,Z -79.114,A 90.000,B 90.000,C 0.000} C_DIS
LIN {X -90.608,Y 21.431,Z -80.110,A 90.000,B 90.000,C 0.000} C_DIS
LIN {X -89.321,Y 21.431,Z -81.056,A 90.000,B 90.000,C 0.000} C_DIS
LIN {X -87.997,Y 21.431,Z -81.950,A 90.000,B 90.000,C 0.000} C_DIS
LIN {X -86.638,Y 21.431,Z -82.790,A 90.000,B 90.000,C 0.000} C_DIS
LIN {X -85.247,Y 21.431,Z -83.576,A 90.000,B 90.000,C 0.000} C_DIS
LIN {X -83.826,Y 21.431,Z -84.305,A 90.000,B 90.000,C 0.000} C_DIS
LIN {X -83.666,Y 21.431,Z -84.379,A 90.000,B 90.000,C 0.000} C_DIS
LIN {X -81.841,Y 21.431,Z -85.125,A 90.000,B 90.000,C 0.000} C_DIS
LIN {X -81.122,Y 21.431,Z -85.328,A 90.000,B 90.000,C 0.000} C_DIS
LIN {X -80.419,Y 21.431,Z -85.583,A 90.000,B 90.000,C 0.000} C_DIS
LIN {X -79.737,Y 21.431,Z -85.888,A 90.000,B 90.000,C 0.000} C_DIS
LIN {X -79.078,Y 21.431,Z -86.242,A 90.000,B 90.000,C 0.000} C_DIS
LIN {X -78.448,Y 21.431,Z -86.644,A 90.000,B 90.000,C 0.000} C_DIS
LIN {X -76.801,Y 21.431,Z -88.072,A 90.000,B 90.000,C 0.000} C_DIS
LIN {X -75.192,Y 21.431,Z -89.542,A 90.000,B 90.000,C 0.000} C_DIS
LIN {X -73.623,Y 21.431,Z -91.055,A 90.000,B 90.000,C 0.000} C_DIS
LIN {X -72.094,Y 21.431,Z -92.608,A 90.000,B 90.000,C 0.000} C_DIS
LIN {X -70.606,Y 21.431,Z -94.201,A 90.000,B 90.000,C 0.000} C_DIS
LIN {X -69.161,Y 21.431,Z -95.833,A 90.000,B 90.000,C 0.000} C_DIS
LIN {X -67.759,Y 21.431,Z -97.502,A 90.000,B 90.000,C 0.000} C_DIS
LIN {X -66.402,Y 21.431,Z -99.208,A 90.000,B 90.000,C 0.000} C_DIS
LIN {X -65.089,Y 21.431,Z -100.948,A 90.000,B 90.000,C 0.000} C_DIS
LIN {X -62.714,Y 21.431,Z -104.281,A 90.000,B 90.000,C 0.000} C_DIS
LIN {X -60.294,Y 21.431,Z -107.582,A 90.000,B 90.000,C 0.000} C_DIS
LIN {X -57.830,Y 21.431,Z -110.851,A 90.000,B 90.000,C 0.000} C_DIS
LIN {X -55.323,Y 21.431,Z -114.085,A 90.000,B 90.000,C 0.000} C_DIS
LIN {X -52.772,Y 21.431,Z -117.286,A 90.000,B 90.000,C 0.000} C_DIS
LIN {X -50.178,Y 21.431,Z -120.452,A 90.000,B 90.000,C 0.000} C_DIS
LIN {X -49.457,Y 21.431,Z -121.220,A 90.000,B 90.000,C 0.000} C_DIS
LIN {X -48.786,Y 21.431,Z -122.033,A 90.000,B 90.000,C 0.000} C_DIS
LIN {X -48.169,Y 21.431,Z -122.887,A 90.000,B 90.000,C 0.000} C_DIS
LIN {X -47.607,Y 21.431,Z -123.778,A 90.000,B 90.000,C 0.000} C_DIS
LIN {X -47.104,Y 21.431,Z -124.704,A 90.000,B 90.000,C 0.000} C_DIS
LIN {X -46.661,Y 21.431,Z -125.660,A 90.000,B 90.000,C 0.000} C_DIS
LIN {X -45.799,Y 21.431,Z -127.912,A 90.000,B 90.000,C 0.000} C_DIS
LIN {X -44.886,Y 21.431,Z -130.143,A 90.000,B 90.000,C 0.000} C_DIS
LIN {X -43.923,Y 21.431,Z -132.354,A 90.000,B 90.000,C 0.000} C_DIS
LIN {X -42.910,Y 21.431,Z -134.542,A 90.000,B 90.000,C 0.000} C_DIS
LIN {X -41.848,Y 21.431,Z -136.706,A 90.000,B 90.000,C 0.000} C_DIS
LIN {X -40.737,Y 21.431,Z -138.846,A 90.000,B 90.000,C 0.000} C_DIS
LIN {X -39.999,Y 21.431,Z -140.200,A 90.000,B 90.000,C 0.000} C_DIS
LIN {X -39.208,Y 21.431,Z -141.524,A 90.000,B 90.000,C 0.000} C_DIS
LIN {X -38.364,Y 21.431,Z -142.815,A 90.000,B 90.000,C 0.000} C_DIS
LIN {X -37.470,Y 21.431,Z -144.071,A 90.000,B 90.000,C 0.000} C_DIS
LIN {X -36.526,Y 21.431,Z -145.291,A 90.000,B 90.000,C 0.000} C_DIS
LIN {X -34.991,Y 21.431,Z -147.109,A 90.000,B 90.000,C 0.000} C_DIS
LIN {X -33.415,Y 21.431,Z -148.892,A 90.000,B 90.000,C 0.000} C_DIS
LIN {X -31.799,Y 21.431,Z -150.639,A 90.000,B 90.000,C 0.000} C_DIS
